	GVL_Modbus.modbusDamperInterface[2][1].enable     := TRUE;
	GVL_Modbus.modbusDamperInterface[2][2].enable     := TRUE;
	GVL_Modbus.modbusDamperInterface[2][3].enable     := TRUE;
	GVL_Modbus.modbusDamperInterface[2][4].enable     := TRUE;
	GVL_Modbus.modbusDamperInterface[2][5].enable     := TRUE;
	GVL_Modbus.modbusDamperInterface[2][6].enable     := TRUE;
	GVL_Modbus.modbusDamperInterface[2][7].enable     := TRUE;
	GVL_Modbus.modbusDamperInterface[2][8].enable     := TRUE;
	GVL_Modbus.modbusDamperInterface[2][9].enable     := TRUE;
	GVL_Modbus.modbusDamperInterface[2][10].enable     := TRUE;
	GVL_Modbus.modbusDamperInterface[2][11].enable     := TRUE;
	GVL_Modbus.modbusDamperInterface[2][12].enable     := TRUE;
	GVL_Modbus.modbusDamperInterface[2][13].enable     := TRUE;
	GVL_Modbus.modbusDamperInterface[2][14].enable     := TRUE;
	GVL_Modbus.modbusDamperInterface[2][15].enable     := TRUE;
	GVL_Modbus.modbusDamperInterface[2][16].enable     := TRUE;
	GVL_Modbus.modbusDamperInterface[2][17].enable     := TRUE;
	GVL_Modbus.modbusDamperInterface[2][18].enable     := TRUE;
	GVL_Modbus.modbusDamperInterface[2][19].enable     := TRUE;
	GVL_Modbus.modbusDamperInterface[2][20].enable     := TRUE;
	GVL_Modbus.modbusDamperInterface[2][21].enable     := TRUE;
	GVL_Modbus.modbusDamperInterface[2][22].enable     := TRUE;
	GVL_Modbus.modbusDamperInterface[2][23].enable     := TRUE;
	GVL_Modbus.modbusDamperInterface[2][24].enable     := TRUE;
	GVL_Modbus.modbusDamperInterface[2][25].enable     := TRUE;
	GVL_Modbus.modbusDamperInterface[2][26].enable     := TRUE;
	GVL_Modbus.modbusDamperInterface[2][1].systemNumber     := 01;
	GVL_Modbus.modbusDamperInterface[2][2].systemNumber     := 01;
	GVL_Modbus.modbusDamperInterface[2][3].systemNumber     := 01;
	GVL_Modbus.modbusDamperInterface[2][4].systemNumber     := 01;
	GVL_Modbus.modbusDamperInterface[2][5].systemNumber     := 01;
	GVL_Modbus.modbusDamperInterface[2][6].systemNumber     := 01;
	GVL_Modbus.modbusDamperInterface[2][7].systemNumber     := 01;
	GVL_Modbus.modbusDamperInterface[2][8].systemNumber     := 01;
	GVL_Modbus.modbusDamperInterface[2][9].systemNumber     := 01;
	GVL_Modbus.modbusDamperInterface[2][10].systemNumber     := 01;
	GVL_Modbus.modbusDamperInterface[2][11].systemNumber     := 01;
	GVL_Modbus.modbusDamperInterface[2][12].systemNumber     := 01;
	GVL_Modbus.modbusDamperInterface[2][13].systemNumber     := 01;
	GVL_Modbus.modbusDamperInterface[2][14].systemNumber     := 01;
	GVL_Modbus.modbusDamperInterface[2][15].systemNumber     := 01;
	GVL_Modbus.modbusDamperInterface[2][16].systemNumber     := 01;
	GVL_Modbus.modbusDamperInterface[2][17].systemNumber     := 01;
	GVL_Modbus.modbusDamperInterface[2][18].systemNumber     := 01;
	GVL_Modbus.modbusDamperInterface[2][19].systemNumber     := 01;
	GVL_Modbus.modbusDamperInterface[2][20].systemNumber     := 01;
	GVL_Modbus.modbusDamperInterface[2][21].systemNumber     := 01;
	GVL_Modbus.modbusDamperInterface[2][22].systemNumber     := 01;
	GVL_Modbus.modbusDamperInterface[2][23].systemNumber     := 01;
	GVL_Modbus.modbusDamperInterface[2][24].systemNumber     := 01;
	GVL_Modbus.modbusDamperInterface[2][25].systemNumber     := 01;
	GVL_Modbus.modbusDamperInterface[2][26].systemNumber     := 01;
	GVL_Modbus.modbusDamperInterface[2][1].systemPrefix     := 'A';
	GVL_Modbus.modbusDamperInterface[2][2].systemPrefix     := 'A';
	GVL_Modbus.modbusDamperInterface[2][3].systemPrefix     := 'A';
	GVL_Modbus.modbusDamperInterface[2][4].systemPrefix     := 'A';
	GVL_Modbus.modbusDamperInterface[2][5].systemPrefix     := 'A';
	GVL_Modbus.modbusDamperInterface[2][6].systemPrefix     := 'A';
	GVL_Modbus.modbusDamperInterface[2][7].systemPrefix     := 'A';
	GVL_Modbus.modbusDamperInterface[2][8].systemPrefix     := 'A';
	GVL_Modbus.modbusDamperInterface[2][9].systemPrefix     := 'A';
	GVL_Modbus.modbusDamperInterface[2][10].systemPrefix     := 'A';
	GVL_Modbus.modbusDamperInterface[2][11].systemPrefix     := 'A';
	GVL_Modbus.modbusDamperInterface[2][12].systemPrefix     := 'A';
	GVL_Modbus.modbusDamperInterface[2][13].systemPrefix     := 'A';
	GVL_Modbus.modbusDamperInterface[2][14].systemPrefix     := 'A';
	GVL_Modbus.modbusDamperInterface[2][15].systemPrefix     := 'A';
	GVL_Modbus.modbusDamperInterface[2][16].systemPrefix     := 'A';
	GVL_Modbus.modbusDamperInterface[2][17].systemPrefix     := 'A';
	GVL_Modbus.modbusDamperInterface[2][18].systemPrefix     := 'A';
	GVL_Modbus.modbusDamperInterface[2][19].systemPrefix     := 'A';
	GVL_Modbus.modbusDamperInterface[2][20].systemPrefix     := 'A';
	GVL_Modbus.modbusDamperInterface[2][21].systemPrefix     := 'A';
	GVL_Modbus.modbusDamperInterface[2][22].systemPrefix     := 'A';
	GVL_Modbus.modbusDamperInterface[2][23].systemPrefix     := 'A';
	GVL_Modbus.modbusDamperInterface[2][24].systemPrefix     := 'A';
	GVL_Modbus.modbusDamperInterface[2][25].systemPrefix     := 'A';
	GVL_Modbus.modbusDamperInterface[2][26].systemPrefix     := 'A';
	GVL_Modbus.modbusDamperInterface[2][1].airDirection     := 1;
	GVL_Modbus.modbusDamperInterface[2][2].airDirection     := 1;
	GVL_Modbus.modbusDamperInterface[2][3].airDirection     := 1;
	GVL_Modbus.modbusDamperInterface[2][4].airDirection     := 0;
	GVL_Modbus.modbusDamperInterface[2][5].airDirection     := 0;
	GVL_Modbus.modbusDamperInterface[2][6].airDirection     := 0;
	GVL_Modbus.modbusDamperInterface[2][7].airDirection     := 1;
	GVL_Modbus.modbusDamperInterface[2][8].airDirection     := 1;
	GVL_Modbus.modbusDamperInterface[2][9].airDirection     := 0;
	GVL_Modbus.modbusDamperInterface[2][10].airDirection     := 0;
	GVL_Modbus.modbusDamperInterface[2][11].airDirection     := 0;
	GVL_Modbus.modbusDamperInterface[2][12].airDirection     := 0;
	GVL_Modbus.modbusDamperInterface[2][13].airDirection     := 0;
	GVL_Modbus.modbusDamperInterface[2][14].airDirection     := 0;
	GVL_Modbus.modbusDamperInterface[2][15].airDirection     := 0;
	GVL_Modbus.modbusDamperInterface[2][16].airDirection     := 0;
	GVL_Modbus.modbusDamperInterface[2][17].airDirection     := 0;
	GVL_Modbus.modbusDamperInterface[2][18].airDirection     := 0;
	GVL_Modbus.modbusDamperInterface[2][19].airDirection     := 0;
	GVL_Modbus.modbusDamperInterface[2][20].airDirection     := 0;
	GVL_Modbus.modbusDamperInterface[2][21].airDirection     := 0;
	GVL_Modbus.modbusDamperInterface[2][22].airDirection     := 0;
	GVL_Modbus.modbusDamperInterface[2][23].airDirection     := 1;
	GVL_Modbus.modbusDamperInterface[2][24].airDirection     := 0;
	GVL_Modbus.modbusDamperInterface[2][25].airDirection     := 0;
	GVL_Modbus.modbusDamperInterface[2][26].airDirection     := 0;
	PersistentVars.ModbusDamperSetpoints[2][3].vMidM3h     := 100;
	PersistentVars.ModbusDamperSetpoints[2][9].vMidM3h     := 100;
	PersistentVars.ModbusDamperSetpoints[2][10].vMidM3h     := 100;
	PersistentVars.ModbusDamperSetpoints[2][11].vMidM3h     := 100;
	PersistentVars.ModbusDamperSetpoints[2][12].vMidM3h     := 100;
	PersistentVars.ModbusDamperSetpoints[2][13].vMidM3h     := 100;
	PersistentVars.ModbusDamperSetpoints[2][14].vMidM3h     := 100;
	PersistentVars.ModbusDamperSetpoints[2][15].vMidM3h     := 100;
	PersistentVars.ModbusDamperSetpoints[2][16].vMidM3h     := 100;
	PersistentVars.ModbusDamperSetpoints[2][17].vMidM3h     := 100;
	PersistentVars.ModbusDamperSetpoints[2][18].vMidM3h     := 160;
	PersistentVars.ModbusDamperSetpoints[2][19].vMidM3h     := 100;
	PersistentVars.ModbusDamperSetpoints[2][20].vMidM3h     := 100;
	PersistentVars.ModbusDamperSetpoints[2][21].vMidM3h     := 100;
	PersistentVars.ModbusDamperSetpoints[2][22].vMidM3h     := 100;
	PersistentVars.ModbusDamperSetpoints[2][24].vMidM3h     := 100;
	PersistentVars.ModbusDamperSetpoints[2][25].vMidM3h     := 100;
	PersistentVars.ModbusDamperSetpoints[2][26].vMidM3h     := 100;
                            
                        
END_ACTION
END_PROGRAM

PROGRAM PRG_DamperLine_3

                
    
	if (firstScan) then
	    initialSettings();
	end_if
	
	GVL_Modbus.modbusDamperInterface[3][1].tag     := 'B=360.02-SQ5UBH1';
	GVL_Modbus.modbusDamperInterface[3][2].tag     := 'B=360.02-SQ5UBH2';
	GVL_Modbus.modbusDamperInterface[3][3].tag     := 'B=360.02-SQ4UBH1';
	GVL_Modbus.modbusDamperInterface[3][4].tag     := 'B=360.02-SQ4UBH2';
	GVL_Modbus.modbusDamperInterface[3][1].damperClimateInterface     := GVL_ClimateControl.typClimateControllerInterfaceRoomSONE.actuators.damper;
	GVL_Modbus.modbusDamperInterface[3][2].damperClimateInterface     := GVL_ClimateControl.typClimateControllerInterfaceRoomSONE.actuators.damper;
	GVL_Modbus.modbusDamperInterface[3][3].damperClimateInterface     := GVL_ClimateControl.typClimateControllerInterfaceRoomSONE.actuators.damper;
	GVL_Modbus.modbusDamperInterface[3][4].damperClimateInterface     := GVL_ClimateControl.typClimateControllerInterfaceRoomSONE.actuators.damper;
                
              

ACTION initialSettings:
                            
                                
	GVL_Modbus.modbusDamperInterface[3][1].enable     := TRUE;
	GVL_Modbus.modbusDamperInterface[3][2].enable     := TRUE;
	GVL_Modbus.modbusDamperInterface[3][3].enable     := TRUE;
	GVL_Modbus.modbusDamperInterface[3][4].enable     := TRUE;
	GVL_Modbus.modbusDamperInterface[3][1].systemNumber     := 02;
	GVL_Modbus.modbusDamperInterface[3][2].systemNumber     := 02;
	GVL_Modbus.modbusDamperInterface[3][3].systemNumber     := 02;
	GVL_Modbus.modbusDamperInterface[3][4].systemNumber     := 02;
	GVL_Modbus.modbusDamperInterface[3][1].systemPrefix     := 'B';
	GVL_Modbus.modbusDamperInterface[3][2].systemPrefix     := 'B';
	GVL_Modbus.modbusDamperInterface[3][3].systemPrefix     := 'B';
	GVL_Modbus.modbusDamperInterface[3][4].systemPrefix     := 'B';
	GVL_Modbus.modbusDamperInterface[3][1].airDirection     := 1;
	GVL_Modbus.modbusDamperInterface[3][2].airDirection     := 1;
	GVL_Modbus.modbusDamperInterface[3][3].airDirection     := 0;
	GVL_Modbus.modbusDamperInterface[3][4].airDirection     := 0;
                            
                        
END_ACTION
END_PROGRAM

PROGRAM PRG_StateTexts

                
    
	IF (firstScan) THEN
C_5640_501_06_RTC01_MOD_FB_R0401.setStateText(1, 'Frostbeskyttelse');
C_5640_501_06_RTC01_MOD_FB_R0401.setStateText(2, 'Økonomi');
C_5640_501_06_RTC01_MOD_FB_R0401.setStateText(3, 'Standby');
C_5640_501_06_RTC01_MOD_FB_R0401.setStateText(4, 'Komfort');
C_5640_501_06_RTC01_MOD_FB_R0401.setStateText(5, 'Nattkjøling');
C_5640_501_06_RTC01_KMD_MSV_R0401.setStateText(1, 'Kalender 1');
C_5640_501_06_RTC01_KMD_MSV_R0401.setStateText(2, 'Kalender 2');
C_5640_501_06_RTC01_KMD_MSV_R0401.setStateText(3, 'Kalender 3');
C_5640_501_06_RTC01_KMD_MSV_R0401.setStateText(4, 'Kalender 4');
C_5640_501_06_RTC01_KMD_MSV_R0401.setStateText(5, 'Kalender 5');
C_5640_501_06_RTC01_KMD_MSV_R0401.setStateText(6, 'Kalender 6');
C_5640_501_06_RTC01_KMD_MSV_R0401.setStateText(7, 'Kalender 7');
C_5640_501_06_RTC01_KMD_MSV_R0401.setStateText(8, 'Kalender 8');
C_5640_501_06_RTC01_KMD_MSV_R0401.setStateText(9, 'Kalender 9');
C_5640_501_06_RTC01_KMD_MSV_R0401.setStateText(10, 'Kalender 10');
C_5640_501_06_RTC01_MOD_FB_R0406.setStateText(1, 'Frostbeskyttelse');
C_5640_501_06_RTC01_MOD_FB_R0406.setStateText(2, 'Økonomi');
C_5640_501_06_RTC01_MOD_FB_R0406.setStateText(3, 'Standby');
C_5640_501_06_RTC01_MOD_FB_R0406.setStateText(4, 'Komfort');
C_5640_501_06_RTC01_MOD_FB_R0406.setStateText(5, 'Nattkjøling');
C_5640_501_06_RTC01_KMD_MSV_R0406.setStateText(1, 'Kalender 1');
C_5640_501_06_RTC01_KMD_MSV_R0406.setStateText(2, 'Kalender 2');
C_5640_501_06_RTC01_KMD_MSV_R0406.setStateText(3, 'Kalender 3');
C_5640_501_06_RTC01_KMD_MSV_R0406.setStateText(4, 'Kalender 4');
C_5640_501_06_RTC01_KMD_MSV_R0406.setStateText(5, 'Kalender 5');
C_5640_501_06_RTC01_KMD_MSV_R0406.setStateText(6, 'Kalender 6');
C_5640_501_06_RTC01_KMD_MSV_R0406.setStateText(7, 'Kalender 7');
C_5640_501_06_RTC01_KMD_MSV_R0406.setStateText(8, 'Kalender 8');
C_5640_501_06_RTC01_KMD_MSV_R0406.setStateText(9, 'Kalender 9');
C_5640_501_06_RTC01_KMD_MSV_R0406.setStateText(10, 'Kalender 10');
C_5640_501_06_RTC01_MOD_FB_R0407.setStateText(1, 'Frostbeskyttelse');
C_5640_501_06_RTC01_MOD_FB_R0407.setStateText(2, 'Økonomi');
C_5640_501_06_RTC01_MOD_FB_R0407.setStateText(3, 'Standby');
C_5640_501_06_RTC01_MOD_FB_R0407.setStateText(4, 'Komfort');
C_5640_501_06_RTC01_MOD_FB_R0407.setStateText(5, 'Nattkjøling');
C_5640_501_06_RTC01_KMD_MSV_R0407.setStateText(1, 'Kalender 1');
C_5640_501_06_RTC01_KMD_MSV_R0407.setStateText(2, 'Kalender 2');
C_5640_501_06_RTC01_KMD_MSV_R0407.setStateText(3, 'Kalender 3');
C_5640_501_06_RTC01_KMD_MSV_R0407.setStateText(4, 'Kalender 4');
C_5640_501_06_RTC01_KMD_MSV_R0407.setStateText(5, 'Kalender 5');
C_5640_501_06_RTC01_KMD_MSV_R0407.setStateText(6, 'Kalender 6');
C_5640_501_06_RTC01_KMD_MSV_R0407.setStateText(7, 'Kalender 7');
C_5640_501_06_RTC01_KMD_MSV_R0407.setStateText(8, 'Kalender 8');
C_5640_501_06_RTC01_KMD_MSV_R0407.setStateText(9, 'Kalender 9');
C_5640_501_06_RTC01_KMD_MSV_R0407.setStateText(10, 'Kalender 10');
C_5640_501_06_RTC01_MOD_FB_R0408.setStateText(1, 'Frostbeskyttelse');
C_5640_501_06_RTC01_MOD_FB_R0408.setStateText(2, 'Økonomi');
C_5640_501_06_RTC01_MOD_FB_R0408.setStateText(3, 'Standby');
C_5640_501_06_RTC01_MOD_FB_R0408.setStateText(4, 'Komfort');
C_5640_501_06_RTC01_MOD_FB_R0408.setStateText(5, 'Nattkjøling');
C_5640_501_06_RTC01_KMD_MSV_R0408.setStateText(1, 'Kalender 1');
C_5640_501_06_RTC01_KMD_MSV_R0408.setStateText(2, 'Kalender 2');
C_5640_501_06_RTC01_KMD_MSV_R0408.setStateText(3, 'Kalender 3');
C_5640_501_06_RTC01_KMD_MSV_R0408.setStateText(4, 'Kalender 4');
C_5640_501_06_RTC01_KMD_MSV_R0408.setStateText(5, 'Kalender 5');
C_5640_501_06_RTC01_KMD_MSV_R0408.setStateText(6, 'Kalender 6');
C_5640_501_06_RTC01_KMD_MSV_R0408.setStateText(7, 'Kalender 7');
C_5640_501_06_RTC01_KMD_MSV_R0408.setStateText(8, 'Kalender 8');
C_5640_501_06_RTC01_KMD_MSV_R0408.setStateText(9, 'Kalender 9');
C_5640_501_06_RTC01_KMD_MSV_R0408.setStateText(10, 'Kalender 10');
C_5640_501_06_RTC01_MOD_FB_R0409.setStateText(1, 'Frostbeskyttelse');
C_5640_501_06_RTC01_MOD_FB_R0409.setStateText(2, 'Økonomi');
C_5640_501_06_RTC01_MOD_FB_R0409.setStateText(3, 'Standby');
C_5640_501_06_RTC01_MOD_FB_R0409.setStateText(4, 'Komfort');
C_5640_501_06_RTC01_MOD_FB_R0409.setStateText(5, 'Nattkjøling');
C_5640_501_06_RTC01_KMD_MSV_R0409.setStateText(1, 'Kalender 1');
C_5640_501_06_RTC01_KMD_MSV_R0409.setStateText(2, 'Kalender 2');
C_5640_501_06_RTC01_KMD_MSV_R0409.setStateText(3, 'Kalender 3');
C_5640_501_06_RTC01_KMD_MSV_R0409.setStateText(4, 'Kalender 4');
C_5640_501_06_RTC01_KMD_MSV_R0409.setStateText(5, 'Kalender 5');
C_5640_501_06_RTC01_KMD_MSV_R0409.setStateText(6, 'Kalender 6');
C_5640_501_06_RTC01_KMD_MSV_R0409.setStateText(7, 'Kalender 7');
C_5640_501_06_RTC01_KMD_MSV_R0409.setStateText(8, 'Kalender 8');
C_5640_501_06_RTC01_KMD_MSV_R0409.setStateText(9, 'Kalender 9');
C_5640_501_06_RTC01_KMD_MSV_R0409.setStateText(10, 'Kalender 10');
C_5640_501_06_RTC01_MOD_FB_R0464.setStateText(1, 'Frostbeskyttelse');
C_5640_501_06_RTC01_MOD_FB_R0464.setStateText(2, 'Økonomi');
C_5640_501_06_RTC01_MOD_FB_R0464.setStateText(3, 'Standby');
C_5640_501_06_RTC01_MOD_FB_R0464.setStateText(4, 'Komfort');
C_5640_501_06_RTC01_MOD_FB_R0464.setStateText(5, 'Nattkjøling');
C_5640_501_06_RTC01_KMD_MSV_R0464.setStateText(1, 'Kalender 1');
C_5640_501_06_RTC01_KMD_MSV_R0464.setStateText(2, 'Kalender 2');
C_5640_501_06_RTC01_KMD_MSV_R0464.setStateText(3, 'Kalender 3');
C_5640_501_06_RTC01_KMD_MSV_R0464.setStateText(4, 'Kalender 4');
C_5640_501_06_RTC01_KMD_MSV_R0464.setStateText(5, 'Kalender 5');
C_5640_501_06_RTC01_KMD_MSV_R0464.setStateText(6, 'Kalender 6');
C_5640_501_06_RTC01_KMD_MSV_R0464.setStateText(7, 'Kalender 7');
C_5640_501_06_RTC01_KMD_MSV_R0464.setStateText(8, 'Kalender 8');
C_5640_501_06_RTC01_KMD_MSV_R0464.setStateText(9, 'Kalender 9');
C_5640_501_06_RTC01_KMD_MSV_R0464.setStateText(10, 'Kalender 10');
C_5640_501_06_RTC01_MOD_FB_R0415.setStateText(1, 'Frostbeskyttelse');
C_5640_501_06_RTC01_MOD_FB_R0415.setStateText(2, 'Økonomi');
C_5640_501_06_RTC01_MOD_FB_R0415.setStateText(3, 'Standby');
C_5640_501_06_RTC01_MOD_FB_R0415.setStateText(4, 'Komfort');
C_5640_501_06_RTC01_MOD_FB_R0415.setStateText(5, 'Nattkjøling');
C_5640_501_06_RTC01_KMD_MSV_R0415.setStateText(1, 'Kalender 1');
C_5640_501_06_RTC01_KMD_MSV_R0415.setStateText(2, 'Kalender 2');
C_5640_501_06_RTC01_KMD_MSV_R0415.setStateText(3, 'Kalender 3');
C_5640_501_06_RTC01_KMD_MSV_R0415.setStateText(4, 'Kalender 4');
C_5640_501_06_RTC01_KMD_MSV_R0415.setStateText(5, 'Kalender 5');
C_5640_501_06_RTC01_KMD_MSV_R0415.setStateText(6, 'Kalender 6');
C_5640_501_06_RTC01_KMD_MSV_R0415.setStateText(7, 'Kalender 7');
C_5640_501_06_RTC01_KMD_MSV_R0415.setStateText(8, 'Kalender 8');
C_5640_501_06_RTC01_KMD_MSV_R0415.setStateText(9, 'Kalender 9');
C_5640_501_06_RTC01_KMD_MSV_R0415.setStateText(10, 'Kalender 10');
C_5640_501_06_RTC01_MOD_FB_R0422.setStateText(1, 'Frostbeskyttelse');
C_5640_501_06_RTC01_MOD_FB_R0422.setStateText(2, 'Økonomi');
C_5640_501_06_RTC01_MOD_FB_R0422.setStateText(3, 'Standby');
C_5640_501_06_RTC01_MOD_FB_R0422.setStateText(4, 'Komfort');
C_5640_501_06_RTC01_MOD_FB_R0422.setStateText(5, 'Nattkjøling');
C_5640_501_06_RTC01_KMD_MSV_R0422.setStateText(1, 'Kalender 1');
C_5640_501_06_RTC01_KMD_MSV_R0422.setStateText(2, 'Kalender 2');
C_5640_501_06_RTC01_KMD_MSV_R0422.setStateText(3, 'Kalender 3');
C_5640_501_06_RTC01_KMD_MSV_R0422.setStateText(4, 'Kalender 4');
C_5640_501_06_RTC01_KMD_MSV_R0422.setStateText(5, 'Kalender 5');
C_5640_501_06_RTC01_KMD_MSV_R0422.setStateText(6, 'Kalender 6');
C_5640_501_06_RTC01_KMD_MSV_R0422.setStateText(7, 'Kalender 7');
C_5640_501_06_RTC01_KMD_MSV_R0422.setStateText(8, 'Kalender 8');
C_5640_501_06_RTC01_KMD_MSV_R0422.setStateText(9, 'Kalender 9');
C_5640_501_06_RTC01_KMD_MSV_R0422.setStateText(10, 'Kalender 10');
C_5640_501_06_RTC01_MOD_FB_R0426_1.setStateText(1, 'Frostbeskyttelse');
C_5640_501_06_RTC01_MOD_FB_R0426_1.setStateText(2, 'Økonomi');
C_5640_501_06_RTC01_MOD_FB_R0426_1.setStateText(3, 'Standby');
C_5640_501_06_RTC01_MOD_FB_R0426_1.setStateText(4, 'Komfort');
C_5640_501_06_RTC01_MOD_FB_R0426_1.setStateText(5, 'Nattkjøling');
C_5640_501_06_RTC01_KMD_MSV_R0426_1.setStateText(1, 'Kalender 1');
C_5640_501_06_RTC01_KMD_MSV_R0426_1.setStateText(2, 'Kalender 2');
C_5640_501_06_RTC01_KMD_MSV_R0426_1.setStateText(3, 'Kalender 3');
C_5640_501_06_RTC01_KMD_MSV_R0426_1.setStateText(4, 'Kalender 4');
C_5640_501_06_RTC01_KMD_MSV_R0426_1.setStateText(5, 'Kalender 5');
C_5640_501_06_RTC01_KMD_MSV_R0426_1.setStateText(6, 'Kalender 6');
C_5640_501_06_RTC01_KMD_MSV_R0426_1.setStateText(7, 'Kalender 7');
C_5640_501_06_RTC01_KMD_MSV_R0426_1.setStateText(8, 'Kalender 8');
C_5640_501_06_RTC01_KMD_MSV_R0426_1.setStateText(9, 'Kalender 9');
C_5640_501_06_RTC01_KMD_MSV_R0426_1.setStateText(10, 'Kalender 10');
C_5640_501_06_RTC01_MOD_FB_R0426_2.setStateText(1, 'Frostbeskyttelse');
C_5640_501_06_RTC01_MOD_FB_R0426_2.setStateText(2, 'Økonomi');
C_5640_501_06_RTC01_MOD_FB_R0426_2.setStateText(3, 'Standby');
C_5640_501_06_RTC01_MOD_FB_R0426_2.setStateText(4, 'Komfort');
C_5640_501_06_RTC01_MOD_FB_R0426_2.setStateText(5, 'Nattkjøling');
C_5640_501_06_RTC01_KMD_MSV_R0426_2.setStateText(1, 'Kalender 1');
C_5640_501_06_RTC01_KMD_MSV_R0426_2.setStateText(2, 'Kalender 2');
C_5640_501_06_RTC01_KMD_MSV_R0426_2.setStateText(3, 'Kalender 3');
C_5640_501_06_RTC01_KMD_MSV_R0426_2.setStateText(4, 'Kalender 4');
C_5640_501_06_RTC01_KMD_MSV_R0426_2.setStateText(5, 'Kalender 5');
C_5640_501_06_RTC01_KMD_MSV_R0426_2.setStateText(6, 'Kalender 6');
C_5640_501_06_RTC01_KMD_MSV_R0426_2.setStateText(7, 'Kalender 7');
C_5640_501_06_RTC01_KMD_MSV_R0426_2.setStateText(8, 'Kalender 8');
C_5640_501_06_RTC01_KMD_MSV_R0426_2.setStateText(9, 'Kalender 9');
C_5640_501_06_RTC01_KMD_MSV_R0426_2.setStateText(10, 'Kalender 10');
C_5640_501_06_RTC01_MOD_FB_R0426_3.setStateText(1, 'Frostbeskyttelse');
C_5640_501_06_RTC01_MOD_FB_R0426_3.setStateText(2, 'Økonomi');
C_5640_501_06_RTC01_MOD_FB_R0426_3.setStateText(3, 'Standby');
C_5640_501_06_RTC01_MOD_FB_R0426_3.setStateText(4, 'Komfort');
C_5640_501_06_RTC01_MOD_FB_R0426_3.setStateText(5, 'Nattkjøling');
C_5640_501_06_RTC01_KMD_MSV_R0426_3.setStateText(1, 'Kalender 1');
C_5640_501_06_RTC01_KMD_MSV_R0426_3.setStateText(2, 'Kalender 2');
C_5640_501_06_RTC01_KMD_MSV_R0426_3.setStateText(3, 'Kalender 3');
C_5640_501_06_RTC01_KMD_MSV_R0426_3.setStateText(4, 'Kalender 4');
C_5640_501_06_RTC01_KMD_MSV_R0426_3.setStateText(5, 'Kalender 5');
C_5640_501_06_RTC01_KMD_MSV_R0426_3.setStateText(6, 'Kalender 6');
C_5640_501_06_RTC01_KMD_MSV_R0426_3.setStateText(7, 'Kalender 7');
C_5640_501_06_RTC01_KMD_MSV_R0426_3.setStateText(8, 'Kalender 8');
C_5640_501_06_RTC01_KMD_MSV_R0426_3.setStateText(9, 'Kalender 9');
C_5640_501_06_RTC01_KMD_MSV_R0426_3.setStateText(10, 'Kalender 10');
C_5640_501_06_RTC01_MOD_FB_R0528.setStateText(1, 'Frostbeskyttelse');
C_5640_501_06_RTC01_MOD_FB_R0528.setStateText(2, 'Økonomi');
C_5640_501_06_RTC01_MOD_FB_R0528.setStateText(3, 'Standby');
C_5640_501_06_RTC01_MOD_FB_R0528.setStateText(4, 'Komfort');
C_5640_501_06_RTC01_MOD_FB_R0528.setStateText(5, 'Nattkjøling');
C_5640_501_06_RTC01_KMD_MSV_R0528.setStateText(1, 'Kalender 1');
C_5640_501_06_RTC01_KMD_MSV_R0528.setStateText(2, 'Kalender 2');
C_5640_501_06_RTC01_KMD_MSV_R0528.setStateText(3, 'Kalender 3');
C_5640_501_06_RTC01_KMD_MSV_R0528.setStateText(4, 'Kalender 4');
C_5640_501_06_RTC01_KMD_MSV_R0528.setStateText(5, 'Kalender 5');
C_5640_501_06_RTC01_KMD_MSV_R0528.setStateText(6, 'Kalender 6');
C_5640_501_06_RTC01_KMD_MSV_R0528.setStateText(7, 'Kalender 7');
C_5640_501_06_RTC01_KMD_MSV_R0528.setStateText(8, 'Kalender 8');
C_5640_501_06_RTC01_KMD_MSV_R0528.setStateText(9, 'Kalender 9');
C_5640_501_06_RTC01_KMD_MSV_R0528.setStateText(10, 'Kalender 10');
C_5640_501_06_RTC01_MOD_FB_R0523.setStateText(1, 'Frostbeskyttelse');
C_5640_501_06_RTC01_MOD_FB_R0523.setStateText(2, 'Økonomi');
C_5640_501_06_RTC01_MOD_FB_R0523.setStateText(3, 'Standby');
C_5640_501_06_RTC01_MOD_FB_R0523.setStateText(4, 'Komfort');
C_5640_501_06_RTC01_MOD_FB_R0523.setStateText(5, 'Nattkjøling');
C_5640_501_06_RTC01_KMD_MSV_R0523.setStateText(1, 'Kalender 1');
C_5640_501_06_RTC01_KMD_MSV_R0523.setStateText(2, 'Kalender 2');
C_5640_501_06_RTC01_KMD_MSV_R0523.setStateText(3, 'Kalender 3');
C_5640_501_06_RTC01_KMD_MSV_R0523.setStateText(4, 'Kalender 4');
C_5640_501_06_RTC01_KMD_MSV_R0523.setStateText(5, 'Kalender 5');
C_5640_501_06_RTC01_KMD_MSV_R0523.setStateText(6, 'Kalender 6');
C_5640_501_06_RTC01_KMD_MSV_R0523.setStateText(7, 'Kalender 7');
C_5640_501_06_RTC01_KMD_MSV_R0523.setStateText(8, 'Kalender 8');
C_5640_501_06_RTC01_KMD_MSV_R0523.setStateText(9, 'Kalender 9');
C_5640_501_06_RTC01_KMD_MSV_R0523.setStateText(10, 'Kalender 10');
C_5640_501_06_RTC01_MOD_FB_R0531.setStateText(1, 'Frostbeskyttelse');
C_5640_501_06_RTC01_MOD_FB_R0531.setStateText(2, 'Økonomi');
C_5640_501_06_RTC01_MOD_FB_R0531.setStateText(3, 'Standby');
C_5640_501_06_RTC01_MOD_FB_R0531.setStateText(4, 'Komfort');
C_5640_501_06_RTC01_MOD_FB_R0531.setStateText(5, 'Nattkjøling');
C_5640_501_06_RTC01_KMD_MSV_R0531.setStateText(1, 'Kalender 1');
C_5640_501_06_RTC01_KMD_MSV_R0531.setStateText(2, 'Kalender 2');
C_5640_501_06_RTC01_KMD_MSV_R0531.setStateText(3, 'Kalender 3');
C_5640_501_06_RTC01_KMD_MSV_R0531.setStateText(4, 'Kalender 4');
C_5640_501_06_RTC01_KMD_MSV_R0531.setStateText(5, 'Kalender 5');
C_5640_501_06_RTC01_KMD_MSV_R0531.setStateText(6, 'Kalender 6');
C_5640_501_06_RTC01_KMD_MSV_R0531.setStateText(7, 'Kalender 7');
C_5640_501_06_RTC01_KMD_MSV_R0531.setStateText(8, 'Kalender 8');
C_5640_501_06_RTC01_KMD_MSV_R0531.setStateText(9, 'Kalender 9');
C_5640_501_06_RTC01_KMD_MSV_R0531.setStateText(10, 'Kalender 10');
C_5640_501_06_RTC01_MOD_FB_R0535_1.setStateText(1, 'Frostbeskyttelse');
C_5640_501_06_RTC01_MOD_FB_R0535_1.setStateText(2, 'Økonomi');
C_5640_501_06_RTC01_MOD_FB_R0535_1.setStateText(3, 'Standby');
C_5640_501_06_RTC01_MOD_FB_R0535_1.setStateText(4, 'Komfort');
C_5640_501_06_RTC01_MOD_FB_R0535_1.setStateText(5, 'Nattkjøling');
C_5640_501_06_RTC01_KMD_MSV_R0535_1.setStateText(1, 'Kalender 1');
C_5640_501_06_RTC01_KMD_MSV_R0535_1.setStateText(2, 'Kalender 2');
C_5640_501_06_RTC01_KMD_MSV_R0535_1.setStateText(3, 'Kalender 3');
C_5640_501_06_RTC01_KMD_MSV_R0535_1.setStateText(4, 'Kalender 4');
C_5640_501_06_RTC01_KMD_MSV_R0535_1.setStateText(5, 'Kalender 5');
C_5640_501_06_RTC01_KMD_MSV_R0535_1.setStateText(6, 'Kalender 6');
C_5640_501_06_RTC01_KMD_MSV_R0535_1.setStateText(7, 'Kalender 7');
C_5640_501_06_RTC01_KMD_MSV_R0535_1.setStateText(8, 'Kalender 8');
C_5640_501_06_RTC01_KMD_MSV_R0535_1.setStateText(9, 'Kalender 9');
C_5640_501_06_RTC01_KMD_MSV_R0535_1.setStateText(10, 'Kalender 10');
C_5640_501_06_RTC01_MOD_FB_R0535_2.setStateText(1, 'Frostbeskyttelse');
C_5640_501_06_RTC01_MOD_FB_R0535_2.setStateText(2, 'Økonomi');
C_5640_501_06_RTC01_MOD_FB_R0535_2.setStateText(3, 'Standby');
C_5640_501_06_RTC01_MOD_FB_R0535_2.setStateText(4, 'Komfort');
C_5640_501_06_RTC01_MOD_FB_R0535_2.setStateText(5, 'Nattkjøling');
C_5640_501_06_RTC01_KMD_MSV_R0535_2.setStateText(1, 'Kalender 1');
C_5640_501_06_RTC01_KMD_MSV_R0535_2.setStateText(2, 'Kalender 2');
C_5640_501_06_RTC01_KMD_MSV_R0535_2.setStateText(3, 'Kalender 3');
C_5640_501_06_RTC01_KMD_MSV_R0535_2.setStateText(4, 'Kalender 4');
C_5640_501_06_RTC01_KMD_MSV_R0535_2.setStateText(5, 'Kalender 5');
C_5640_501_06_RTC01_KMD_MSV_R0535_2.setStateText(6, 'Kalender 6');
C_5640_501_06_RTC01_KMD_MSV_R0535_2.setStateText(7, 'Kalender 7');
C_5640_501_06_RTC01_KMD_MSV_R0535_2.setStateText(8, 'Kalender 8');
C_5640_501_06_RTC01_KMD_MSV_R0535_2.setStateText(9, 'Kalender 9');
C_5640_501_06_RTC01_KMD_MSV_R0535_2.setStateText(10, 'Kalender 10');
C_5640_501_06_RTC01_MOD_FB_R0535_3.setStateText(1, 'Frostbeskyttelse');
C_5640_501_06_RTC01_MOD_FB_R0535_3.setStateText(2, 'Økonomi');
C_5640_501_06_RTC01_MOD_FB_R0535_3.setStateText(3, 'Standby');
C_5640_501_06_RTC01_MOD_FB_R0535_3.setStateText(4, 'Komfort');
C_5640_501_06_RTC01_MOD_FB_R0535_3.setStateText(5, 'Nattkjøling');
C_5640_501_06_RTC01_KMD_MSV_R0535_3.setStateText(1, 'Kalender 1');
C_5640_501_06_RTC01_KMD_MSV_R0535_3.setStateText(2, 'Kalender 2');
C_5640_501_06_RTC01_KMD_MSV_R0535_3.setStateText(3, 'Kalender 3');
C_5640_501_06_RTC01_KMD_MSV_R0535_3.setStateText(4, 'Kalender 4');
C_5640_501_06_RTC01_KMD_MSV_R0535_3.setStateText(5, 'Kalender 5');
C_5640_501_06_RTC01_KMD_MSV_R0535_3.setStateText(6, 'Kalender 6');
C_5640_501_06_RTC01_KMD_MSV_R0535_3.setStateText(7, 'Kalender 7');
C_5640_501_06_RTC01_KMD_MSV_R0535_3.setStateText(8, 'Kalender 8');
C_5640_501_06_RTC01_KMD_MSV_R0535_3.setStateText(9, 'Kalender 9');
C_5640_501_06_RTC01_KMD_MSV_R0535_3.setStateText(10, 'Kalender 10');
C_5640_501_06_RTC01_MOD_FB_R0536.setStateText(1, 'Frostbeskyttelse');
C_5640_501_06_RTC01_MOD_FB_R0536.setStateText(2, 'Økonomi');
C_5640_501_06_RTC01_MOD_FB_R0536.setStateText(3, 'Standby');
C_5640_501_06_RTC01_MOD_FB_R0536.setStateText(4, 'Komfort');
C_5640_501_06_RTC01_MOD_FB_R0536.setStateText(5, 'Nattkjøling');
C_5640_501_06_RTC01_KMD_MSV_R0536.setStateText(1, 'Kalender 1');
C_5640_501_06_RTC01_KMD_MSV_R0536.setStateText(2, 'Kalender 2');
C_5640_501_06_RTC01_KMD_MSV_R0536.setStateText(3, 'Kalender 3');
C_5640_501_06_RTC01_KMD_MSV_R0536.setStateText(4, 'Kalender 4');
C_5640_501_06_RTC01_KMD_MSV_R0536.setStateText(5, 'Kalender 5');
C_5640_501_06_RTC01_KMD_MSV_R0536.setStateText(6, 'Kalender 6');
C_5640_501_06_RTC01_KMD_MSV_R0536.setStateText(7, 'Kalender 7');
C_5640_501_06_RTC01_KMD_MSV_R0536.setStateText(8, 'Kalender 8');
C_5640_501_06_RTC01_KMD_MSV_R0536.setStateText(9, 'Kalender 9');
C_5640_501_06_RTC01_KMD_MSV_R0536.setStateText(10, 'Kalender 10');
C_5640_501_06_RTC01_MOD_FB_R0543.setStateText(1, 'Frostbeskyttelse');
C_5640_501_06_RTC01_MOD_FB_R0543.setStateText(2, 'Økonomi');
C_5640_501_06_RTC01_MOD_FB_R0543.setStateText(3, 'Standby');
C_5640_501_06_RTC01_MOD_FB_R0543.setStateText(4, 'Komfort');
C_5640_501_06_RTC01_MOD_FB_R0543.setStateText(5, 'Nattkjøling');
C_5640_501_06_RTC01_KMD_MSV_R0543.setStateText(1, 'Kalender 1');
C_5640_501_06_RTC01_KMD_MSV_R0543.setStateText(2, 'Kalender 2');
C_5640_501_06_RTC01_KMD_MSV_R0543.setStateText(3, 'Kalender 3');
C_5640_501_06_RTC01_KMD_MSV_R0543.setStateText(4, 'Kalender 4');
C_5640_501_06_RTC01_KMD_MSV_R0543.setStateText(5, 'Kalender 5');
C_5640_501_06_RTC01_KMD_MSV_R0543.setStateText(6, 'Kalender 6');
C_5640_501_06_RTC01_KMD_MSV_R0543.setStateText(7, 'Kalender 7');
C_5640_501_06_RTC01_KMD_MSV_R0543.setStateText(8, 'Kalender 8');
C_5640_501_06_RTC01_KMD_MSV_R0543.setStateText(9, 'Kalender 9');
C_5640_501_06_RTC01_KMD_MSV_R0543.setStateText(10, 'Kalender 10');
C_5640_501_06_RTC01_MOD_FB_R0547_1.setStateText(1, 'Frostbeskyttelse');
C_5640_501_06_RTC01_MOD_FB_R0547_1.setStateText(2, 'Økonomi');
C_5640_501_06_RTC01_MOD_FB_R0547_1.setStateText(3, 'Standby');
C_5640_501_06_RTC01_MOD_FB_R0547_1.setStateText(4, 'Komfort');
C_5640_501_06_RTC01_MOD_FB_R0547_1.setStateText(5, 'Nattkjøling');
C_5640_501_06_RTC01_KMD_MSV_R0547_1.setStateText(1, 'Kalender 1');
C_5640_501_06_RTC01_KMD_MSV_R0547_1.setStateText(2, 'Kalender 2');
C_5640_501_06_RTC01_KMD_MSV_R0547_1.setStateText(3, 'Kalender 3');
C_5640_501_06_RTC01_KMD_MSV_R0547_1.setStateText(4, 'Kalender 4');
C_5640_501_06_RTC01_KMD_MSV_R0547_1.setStateText(5, 'Kalender 5');
C_5640_501_06_RTC01_KMD_MSV_R0547_1.setStateText(6, 'Kalender 6');
C_5640_501_06_RTC01_KMD_MSV_R0547_1.setStateText(7, 'Kalender 7');
C_5640_501_06_RTC01_KMD_MSV_R0547_1.setStateText(8, 'Kalender 8');
C_5640_501_06_RTC01_KMD_MSV_R0547_1.setStateText(9, 'Kalender 9');
C_5640_501_06_RTC01_KMD_MSV_R0547_1.setStateText(10, 'Kalender 10');
C_5640_501_06_RTC01_MOD_FB_R0547_2.setStateText(1, 'Frostbeskyttelse');
C_5640_501_06_RTC01_MOD_FB_R0547_2.setStateText(2, 'Økonomi');
C_5640_501_06_RTC01_MOD_FB_R0547_2.setStateText(3, 'Standby');
C_5640_501_06_RTC01_MOD_FB_R0547_2.setStateText(4, 'Komfort');
C_5640_501_06_RTC01_MOD_FB_R0547_2.setStateText(5, 'Nattkjøling');
C_5640_501_06_RTC01_KMD_MSV_R0547_2.setStateText(1, 'Kalender 1');
C_5640_501_06_RTC01_KMD_MSV_R0547_2.setStateText(2, 'Kalender 2');
C_5640_501_06_RTC01_KMD_MSV_R0547_2.setStateText(3, 'Kalender 3');
C_5640_501_06_RTC01_KMD_MSV_R0547_2.setStateText(4, 'Kalender 4');
C_5640_501_06_RTC01_KMD_MSV_R0547_2.setStateText(5, 'Kalender 5');
C_5640_501_06_RTC01_KMD_MSV_R0547_2.setStateText(6, 'Kalender 6');
C_5640_501_06_RTC01_KMD_MSV_R0547_2.setStateText(7, 'Kalender 7');
C_5640_501_06_RTC01_KMD_MSV_R0547_2.setStateText(8, 'Kalender 8');
C_5640_501_06_RTC01_KMD_MSV_R0547_2.setStateText(9, 'Kalender 9');
C_5640_501_06_RTC01_KMD_MSV_R0547_2.setStateText(10, 'Kalender 10');
C_5640_501_06_RTC01_MOD_FB_R0544.setStateText(1, 'Frostbeskyttelse');
C_5640_501_06_RTC01_MOD_FB_R0544.setStateText(2, 'Økonomi');
C_5640_501_06_RTC01_MOD_FB_R0544.setStateText(3, 'Standby');
C_5640_501_06_RTC01_MOD_FB_R0544.setStateText(4, 'Komfort');
C_5640_501_06_RTC01_MOD_FB_R0544.setStateText(5, 'Nattkjøling');
C_5640_501_06_RTC01_KMD_MSV_R0544.setStateText(1, 'Kalender 1');
C_5640_501_06_RTC01_KMD_MSV_R0544.setStateText(2, 'Kalender 2');
C_5640_501_06_RTC01_KMD_MSV_R0544.setStateText(3, 'Kalender 3');
C_5640_501_06_RTC01_KMD_MSV_R0544.setStateText(4, 'Kalender 4');
C_5640_501_06_RTC01_KMD_MSV_R0544.setStateText(5, 'Kalender 5');
C_5640_501_06_RTC01_KMD_MSV_R0544.setStateText(6, 'Kalender 6');
C_5640_501_06_RTC01_KMD_MSV_R0544.setStateText(7, 'Kalender 7');
C_5640_501_06_RTC01_KMD_MSV_R0544.setStateText(8, 'Kalender 8');
C_5640_501_06_RTC01_KMD_MSV_R0544.setStateText(9, 'Kalender 9');
C_5640_501_06_RTC01_KMD_MSV_R0544.setStateText(10, 'Kalender 10');
A_360_01_SQ4_A407_KMD.setStateText(1, 'Auto');
A_360_01_SQ4_A407_KMD.setStateText(2, 'Åpne');
A_360_01_SQ4_A407_KMD.setStateText(3, 'Lukke');
A_360_01_SQ4_A407_KMD.setStateText(4, 'Til minste luftmengde');
A_360_01_SQ4_A407_KMD.setStateText(5, 'Til midterste luftmengde');
A_360_01_SQ4_A407_KMD.setStateText(6, 'Til største luftmengde');
A_360_01_SQ4_A407_KMD.setStateText(7, 'Åpne (rask)');
A_360_01_SQ4_A407_KMD.setStateText(8, 'Lukke (rask)');
A_360_01_SQ4_4AH2_KMD.setStateText(1, 'Auto');
A_360_01_SQ4_4AH2_KMD.setStateText(2, 'Åpne');
A_360_01_SQ4_4AH2_KMD.setStateText(3, 'Lukke');
A_360_01_SQ4_4AH2_KMD.setStateText(4, 'Til minste luftmengde');
A_360_01_SQ4_4AH2_KMD.setStateText(5, 'Til midterste luftmengde');
A_360_01_SQ4_4AH2_KMD.setStateText(6, 'Til største luftmengde');
A_360_01_SQ4_4AH2_KMD.setStateText(7, 'Åpne (rask)');
A_360_01_SQ4_4AH2_KMD.setStateText(8, 'Lukke (rask)');
A_360_01_SQ4_4AH1_KMD.setStateText(1, 'Auto');
A_360_01_SQ4_4AH1_KMD.setStateText(2, 'Åpne');
A_360_01_SQ4_4AH1_KMD.setStateText(3, 'Lukke');
A_360_01_SQ4_4AH1_KMD.setStateText(4, 'Til minste luftmengde');
A_360_01_SQ4_4AH1_KMD.setStateText(5, 'Til midterste luftmengde');
A_360_01_SQ4_4AH1_KMD.setStateText(6, 'Til største luftmengde');
A_360_01_SQ4_4AH1_KMD.setStateText(7, 'Åpne (rask)');
A_360_01_SQ4_4AH1_KMD.setStateText(8, 'Lukke (rask)');
A_360_01_SQ5_4AH1_KMD.setStateText(1, 'Auto');
A_360_01_SQ5_4AH1_KMD.setStateText(2, 'Åpne');
A_360_01_SQ5_4AH1_KMD.setStateText(3, 'Lukke');
A_360_01_SQ5_4AH1_KMD.setStateText(4, 'Til minste luftmengde');
A_360_01_SQ5_4AH1_KMD.setStateText(5, 'Til midterste luftmengde');
A_360_01_SQ5_4AH1_KMD.setStateText(6, 'Til største luftmengde');
A_360_01_SQ5_4AH1_KMD.setStateText(7, 'Åpne (rask)');
A_360_01_SQ5_4AH1_KMD.setStateText(8, 'Lukke (rask)');
A_360_01_SQ5_A405_KMD.setStateText(1, 'Auto');
A_360_01_SQ5_A405_KMD.setStateText(2, 'Åpne');
A_360_01_SQ5_A405_KMD.setStateText(3, 'Lukke');
A_360_01_SQ5_A405_KMD.setStateText(4, 'Til minste luftmengde');
A_360_01_SQ5_A405_KMD.setStateText(5, 'Til midterste luftmengde');
A_360_01_SQ5_A405_KMD.setStateText(6, 'Til største luftmengde');
A_360_01_SQ5_A405_KMD.setStateText(7, 'Åpne (rask)');
A_360_01_SQ5_A405_KMD.setStateText(8, 'Lukke (rask)');
A_360_01_SQ4_A401_2_KMD.setStateText(1, 'Auto');
A_360_01_SQ4_A401_2_KMD.setStateText(2, 'Åpne');
A_360_01_SQ4_A401_2_KMD.setStateText(3, 'Lukke');
A_360_01_SQ4_A401_2_KMD.setStateText(4, 'Til minste luftmengde');
A_360_01_SQ4_A401_2_KMD.setStateText(5, 'Til midterste luftmengde');
A_360_01_SQ4_A401_2_KMD.setStateText(6, 'Til største luftmengde');
A_360_01_SQ4_A401_2_KMD.setStateText(7, 'Åpne (rask)');
A_360_01_SQ4_A401_2_KMD.setStateText(8, 'Lukke (rask)');
A_360_01_SQ4_A401_1_KMD.setStateText(1, 'Auto');
A_360_01_SQ4_A401_1_KMD.setStateText(2, 'Åpne');
A_360_01_SQ4_A401_1_KMD.setStateText(3, 'Lukke');
A_360_01_SQ4_A401_1_KMD.setStateText(4, 'Til minste luftmengde');
A_360_01_SQ4_A401_1_KMD.setStateText(5, 'Til midterste luftmengde');
A_360_01_SQ4_A401_1_KMD.setStateText(6, 'Til største luftmengde');
A_360_01_SQ4_A401_1_KMD.setStateText(7, 'Åpne (rask)');
A_360_01_SQ4_A401_1_KMD.setStateText(8, 'Lukke (rask)');
A_360_01_SQ4_A401_KMD.setStateText(1, 'Auto');
A_360_01_SQ4_A401_KMD.setStateText(2, 'Åpne');
A_360_01_SQ4_A401_KMD.setStateText(3, 'Lukke');
A_360_01_SQ4_A401_KMD.setStateText(4, 'Til minste luftmengde');
A_360_01_SQ4_A401_KMD.setStateText(5, 'Til midterste luftmengde');
A_360_01_SQ4_A401_KMD.setStateText(6, 'Til største luftmengde');
A_360_01_SQ4_A401_KMD.setStateText(7, 'Åpne (rask)');
A_360_01_SQ4_A401_KMD.setStateText(8, 'Lukke (rask)');
A_360_01_SQ4_A406_KMD.setStateText(1, 'Auto');
A_360_01_SQ4_A406_KMD.setStateText(2, 'Åpne');
A_360_01_SQ4_A406_KMD.setStateText(3, 'Lukke');
A_360_01_SQ4_A406_KMD.setStateText(4, 'Til minste luftmengde');
A_360_01_SQ4_A406_KMD.setStateText(5, 'Til midterste luftmengde');
A_360_01_SQ4_A406_KMD.setStateText(6, 'Til største luftmengde');
A_360_01_SQ4_A406_KMD.setStateText(7, 'Åpne (rask)');
A_360_01_SQ4_A406_KMD.setStateText(8, 'Lukke (rask)');
A_360_01_SQ4_A408_KMD.setStateText(1, 'Auto');
A_360_01_SQ4_A408_KMD.setStateText(2, 'Åpne');
A_360_01_SQ4_A408_KMD.setStateText(3, 'Lukke');
A_360_01_SQ4_A408_KMD.setStateText(4, 'Til minste luftmengde');
A_360_01_SQ4_A408_KMD.setStateText(5, 'Til midterste luftmengde');
A_360_01_SQ4_A408_KMD.setStateText(6, 'Til største luftmengde');
A_360_01_SQ4_A408_KMD.setStateText(7, 'Åpne (rask)');
A_360_01_SQ4_A408_KMD.setStateText(8, 'Lukke (rask)');
A_360_01_SQ4_A410_1_KMD.setStateText(1, 'Auto');
A_360_01_SQ4_A410_1_KMD.setStateText(2, 'Åpne');
A_360_01_SQ4_A410_1_KMD.setStateText(3, 'Lukke');
A_360_01_SQ4_A410_1_KMD.setStateText(4, 'Til minste luftmengde');
A_360_01_SQ4_A410_1_KMD.setStateText(5, 'Til midterste luftmengde');
A_360_01_SQ4_A410_1_KMD.setStateText(6, 'Til største luftmengde');
A_360_01_SQ4_A410_1_KMD.setStateText(7, 'Åpne (rask)');
A_360_01_SQ4_A410_1_KMD.setStateText(8, 'Lukke (rask)');
A_360_01_SQ4_A410_2_KMD.setStateText(1, 'Auto');
A_360_01_SQ4_A410_2_KMD.setStateText(2, 'Åpne');
A_360_01_SQ4_A410_2_KMD.setStateText(3, 'Lukke');
A_360_01_SQ4_A410_2_KMD.setStateText(4, 'Til minste luftmengde');
A_360_01_SQ4_A410_2_KMD.setStateText(5, 'Til midterste luftmengde');
A_360_01_SQ4_A410_2_KMD.setStateText(6, 'Til største luftmengde');
A_360_01_SQ4_A410_2_KMD.setStateText(7, 'Åpne (rask)');
A_360_01_SQ4_A410_2_KMD.setStateText(8, 'Lukke (rask)');
A_360_01_SQ4_A410_3_KMD.setStateText(1, 'Auto');
A_360_01_SQ4_A410_3_KMD.setStateText(2, 'Åpne');
A_360_01_SQ4_A410_3_KMD.setStateText(3, 'Lukke');
A_360_01_SQ4_A410_3_KMD.setStateText(4, 'Til minste luftmengde');
A_360_01_SQ4_A410_3_KMD.setStateText(5, 'Til midterste luftmengde');
A_360_01_SQ4_A410_3_KMD.setStateText(6, 'Til største luftmengde');
A_360_01_SQ4_A410_3_KMD.setStateText(7, 'Åpne (rask)');
A_360_01_SQ4_A410_3_KMD.setStateText(8, 'Lukke (rask)');
A_360_01_SQ4_A410_4_KMD.setStateText(1, 'Auto');
A_360_01_SQ4_A410_4_KMD.setStateText(2, 'Åpne');
A_360_01_SQ4_A410_4_KMD.setStateText(3, 'Lukke');
A_360_01_SQ4_A410_4_KMD.setStateText(4, 'Til minste luftmengde');
A_360_01_SQ4_A410_4_KMD.setStateText(5, 'Til midterste luftmengde');
A_360_01_SQ4_A410_4_KMD.setStateText(6, 'Til største luftmengde');
A_360_01_SQ4_A410_4_KMD.setStateText(7, 'Åpne (rask)');
A_360_01_SQ4_A410_4_KMD.setStateText(8, 'Lukke (rask)');
A_360_01_SQ4_A410_5_KMD.setStateText(1, 'Auto');
A_360_01_SQ4_A410_5_KMD.setStateText(2, 'Åpne');
A_360_01_SQ4_A410_5_KMD.setStateText(3, 'Lukke');
A_360_01_SQ4_A410_5_KMD.setStateText(4, 'Til minste luftmengde');
A_360_01_SQ4_A410_5_KMD.setStateText(5, 'Til midterste luftmengde');
A_360_01_SQ4_A410_5_KMD.setStateText(6, 'Til største luftmengde');
A_360_01_SQ4_A410_5_KMD.setStateText(7, 'Åpne (rask)');
A_360_01_SQ4_A410_5_KMD.setStateText(8, 'Lukke (rask)');
A_360_01_SQ4_A412_KMD.setStateText(1, 'Auto');
A_360_01_SQ4_A412_KMD.setStateText(2, 'Åpne');
A_360_01_SQ4_A412_KMD.setStateText(3, 'Lukke');
A_360_01_SQ4_A412_KMD.setStateText(4, 'Til minste luftmengde');
A_360_01_SQ4_A412_KMD.setStateText(5, 'Til midterste luftmengde');
A_360_01_SQ4_A412_KMD.setStateText(6, 'Til største luftmengde');
A_360_01_SQ4_A412_KMD.setStateText(7, 'Åpne (rask)');
A_360_01_SQ4_A412_KMD.setStateText(8, 'Lukke (rask)');
A_360_01_SQ4_A413_KMD.setStateText(1, 'Auto');
A_360_01_SQ4_A413_KMD.setStateText(2, 'Åpne');
A_360_01_SQ4_A413_KMD.setStateText(3, 'Lukke');
A_360_01_SQ4_A413_KMD.setStateText(4, 'Til minste luftmengde');
A_360_01_SQ4_A413_KMD.setStateText(5, 'Til midterste luftmengde');
A_360_01_SQ4_A413_KMD.setStateText(6, 'Til største luftmengde');
A_360_01_SQ4_A413_KMD.setStateText(7, 'Åpne (rask)');
A_360_01_SQ4_A413_KMD.setStateText(8, 'Lukke (rask)');
A_360_01_SK4_A415_KMD.setStateText(1, 'Auto');
A_360_01_SK4_A415_KMD.setStateText(2, 'Åpne');
A_360_01_SK4_A415_KMD.setStateText(3, 'Lukke');
A_360_01_SK4_A415_KMD.setStateText(4, 'Til minste luftmengde');
A_360_01_SK4_A415_KMD.setStateText(5, 'Til midterste luftmengde');
A_360_01_SK4_A415_KMD.setStateText(6, 'Til største luftmengde');
A_360_01_SK4_A415_KMD.setStateText(7, 'Åpne (rask)');
A_360_01_SK4_A415_KMD.setStateText(8, 'Lukke (rask)');
A_360_01_SK5_A415_KMD.setStateText(1, 'Auto');
A_360_01_SK5_A415_KMD.setStateText(2, 'Åpne');
A_360_01_SK5_A415_KMD.setStateText(3, 'Lukke');
A_360_01_SK5_A415_KMD.setStateText(4, 'Til minste luftmengde');
A_360_01_SK5_A415_KMD.setStateText(5, 'Til midterste luftmengde');
A_360_01_SK5_A415_KMD.setStateText(6, 'Til største luftmengde');
A_360_01_SK5_A415_KMD.setStateText(7, 'Åpne (rask)');
A_360_01_SK5_A415_KMD.setStateText(8, 'Lukke (rask)');
A_360_01_SK5_A418_KMD.setStateText(1, 'Auto');
A_360_01_SK5_A418_KMD.setStateText(2, 'Åpne');
A_360_01_SK5_A418_KMD.setStateText(3, 'Lukke');
A_360_01_SK5_A418_KMD.setStateText(4, 'Til minste luftmengde');
A_360_01_SK5_A418_KMD.setStateText(5, 'Til midterste luftmengde');
A_360_01_SK5_A418_KMD.setStateText(6, 'Til største luftmengde');
A_360_01_SK5_A418_KMD.setStateText(7, 'Åpne (rask)');
A_360_01_SK5_A418_KMD.setStateText(8, 'Lukke (rask)');
A_360_01_SK4_A417_KMD.setStateText(1, 'Auto');
A_360_01_SK4_A417_KMD.setStateText(2, 'Åpne');
A_360_01_SK4_A417_KMD.setStateText(3, 'Lukke');
A_360_01_SK4_A417_KMD.setStateText(4, 'Til minste luftmengde');
A_360_01_SK4_A417_KMD.setStateText(5, 'Til midterste luftmengde');
A_360_01_SK4_A417_KMD.setStateText(6, 'Til største luftmengde');
A_360_01_SK4_A417_KMD.setStateText(7, 'Åpne (rask)');
A_360_01_SK4_A417_KMD.setStateText(8, 'Lukke (rask)');
A_360_01_SQ5_C411_KMD.setStateText(1, 'Auto');
A_360_01_SQ5_C411_KMD.setStateText(2, 'Åpne');
A_360_01_SQ5_C411_KMD.setStateText(3, 'Lukke');
A_360_01_SQ5_C411_KMD.setStateText(4, 'Til minste luftmengde');
A_360_01_SQ5_C411_KMD.setStateText(5, 'Til midterste luftmengde');
A_360_01_SQ5_C411_KMD.setStateText(6, 'Til største luftmengde');
A_360_01_SQ5_C411_KMD.setStateText(7, 'Åpne (rask)');
A_360_01_SQ5_C411_KMD.setStateText(8, 'Lukke (rask)');
A_360_01_SK5_A421_KMD.setStateText(1, 'Auto');
A_360_01_SK5_A421_KMD.setStateText(2, 'Åpne');
A_360_01_SK5_A421_KMD.setStateText(3, 'Lukke');
A_360_01_SK5_A421_KMD.setStateText(4, 'Til minste luftmengde');
A_360_01_SK5_A421_KMD.setStateText(5, 'Til midterste luftmengde');
A_360_01_SK5_A421_KMD.setStateText(6, 'Til største luftmengde');
A_360_01_SK5_A421_KMD.setStateText(7, 'Åpne (rask)');
A_360_01_SK5_A421_KMD.setStateText(8, 'Lukke (rask)');
A_360_01_SQ5_4AH2_KMD.setStateText(1, 'Auto');
A_360_01_SQ5_4AH2_KMD.setStateText(2, 'Åpne');
A_360_01_SQ5_4AH2_KMD.setStateText(3, 'Lukke');
A_360_01_SQ5_4AH2_KMD.setStateText(4, 'Til minste luftmengde');
A_360_01_SQ5_4AH2_KMD.setStateText(5, 'Til midterste luftmengde');
A_360_01_SQ5_4AH2_KMD.setStateText(6, 'Til største luftmengde');
A_360_01_SQ5_4AH2_KMD.setStateText(7, 'Åpne (rask)');
A_360_01_SQ5_4AH2_KMD.setStateText(8, 'Lukke (rask)');
A_360_01_SK5_A424_KMD.setStateText(1, 'Auto');
A_360_01_SK5_A424_KMD.setStateText(2, 'Åpne');
A_360_01_SK5_A424_KMD.setStateText(3, 'Lukke');
A_360_01_SK5_A424_KMD.setStateText(4, 'Til minste luftmengde');
A_360_01_SK5_A424_KMD.setStateText(5, 'Til midterste luftmengde');
A_360_01_SK5_A424_KMD.setStateText(6, 'Til største luftmengde');
A_360_01_SK5_A424_KMD.setStateText(7, 'Åpne (rask)');
A_360_01_SK5_A424_KMD.setStateText(8, 'Lukke (rask)');
A_360_01_SQ4_4AH3_KMD.setStateText(1, 'Auto');
A_360_01_SQ4_4AH3_KMD.setStateText(2, 'Åpne');
A_360_01_SQ4_4AH3_KMD.setStateText(3, 'Lukke');
A_360_01_SQ4_4AH3_KMD.setStateText(4, 'Til minste luftmengde');
A_360_01_SQ4_4AH3_KMD.setStateText(5, 'Til midterste luftmengde');
A_360_01_SQ4_4AH3_KMD.setStateText(6, 'Til største luftmengde');
A_360_01_SQ4_4AH3_KMD.setStateText(7, 'Åpne (rask)');
A_360_01_SQ4_4AH3_KMD.setStateText(8, 'Lukke (rask)');
A_360_01_SQ4_4AH4_KMD.setStateText(1, 'Auto');
A_360_01_SQ4_4AH4_KMD.setStateText(2, 'Åpne');
A_360_01_SQ4_4AH4_KMD.setStateText(3, 'Lukke');
A_360_01_SQ4_4AH4_KMD.setStateText(4, 'Til minste luftmengde');
A_360_01_SQ4_4AH4_KMD.setStateText(5, 'Til midterste luftmengde');
A_360_01_SQ4_4AH4_KMD.setStateText(6, 'Til største luftmengde');
A_360_01_SQ4_4AH4_KMD.setStateText(7, 'Åpne (rask)');
A_360_01_SQ4_4AH4_KMD.setStateText(8, 'Lukke (rask)');
A_360_01_SQ4_4AH5_KMD.setStateText(1, 'Auto');
A_360_01_SQ4_4AH5_KMD.setStateText(2, 'Åpne');
A_360_01_SQ4_4AH5_KMD.setStateText(3, 'Lukke');
A_360_01_SQ4_4AH5_KMD.setStateText(4, 'Til minste luftmengde');
A_360_01_SQ4_4AH5_KMD.setStateText(5, 'Til midterste luftmengde');
A_360_01_SQ4_4AH5_KMD.setStateText(6, 'Til største luftmengde');
A_360_01_SQ4_4AH5_KMD.setStateText(7, 'Åpne (rask)');
A_360_01_SQ4_4AH5_KMD.setStateText(8, 'Lukke (rask)');
A_360_01_SQ5_4AH3_KMD.setStateText(1, 'Auto');
A_360_01_SQ5_4AH3_KMD.setStateText(2, 'Åpne');
A_360_01_SQ5_4AH3_KMD.setStateText(3, 'Lukke');
A_360_01_SQ5_4AH3_KMD.setStateText(4, 'Til minste luftmengde');
A_360_01_SQ5_4AH3_KMD.setStateText(5, 'Til midterste luftmengde');
A_360_01_SQ5_4AH3_KMD.setStateText(6, 'Til største luftmengde');
A_360_01_SQ5_4AH3_KMD.setStateText(7, 'Åpne (rask)');
A_360_01_SQ5_4AH3_KMD.setStateText(8, 'Lukke (rask)');
A_360_01_SQ5_A401_KMD.setStateText(1, 'Auto');
A_360_01_SQ5_A401_KMD.setStateText(2, 'Åpne');
A_360_01_SQ5_A401_KMD.setStateText(3, 'Lukke');
A_360_01_SQ5_A401_KMD.setStateText(4, 'Til minste luftmengde');
A_360_01_SQ5_A401_KMD.setStateText(5, 'Til midterste luftmengde');
A_360_01_SQ5_A401_KMD.setStateText(6, 'Til største luftmengde');
A_360_01_SQ5_A401_KMD.setStateText(7, 'Åpne (rask)');
A_360_01_SQ5_A401_KMD.setStateText(8, 'Lukke (rask)');
A_360_01_SQ4_A403_KMD.setStateText(1, 'Auto');
A_360_01_SQ4_A403_KMD.setStateText(2, 'Åpne');
A_360_01_SQ4_A403_KMD.setStateText(3, 'Lukke');
A_360_01_SQ4_A403_KMD.setStateText(4, 'Til minste luftmengde');
A_360_01_SQ4_A403_KMD.setStateText(5, 'Til midterste luftmengde');
A_360_01_SQ4_A403_KMD.setStateText(6, 'Til største luftmengde');
A_360_01_SQ4_A403_KMD.setStateText(7, 'Åpne (rask)');
A_360_01_SQ4_A403_KMD.setStateText(8, 'Lukke (rask)');
A_360_01_SQ4_A401_3_KMD.setStateText(1, 'Auto');
A_360_01_SQ4_A401_3_KMD.setStateText(2, 'Åpne');
A_360_01_SQ4_A401_3_KMD.setStateText(3, 'Lukke');
A_360_01_SQ4_A401_3_KMD.setStateText(4, 'Til minste luftmengde');
A_360_01_SQ4_A401_3_KMD.setStateText(5, 'Til midterste luftmengde');
A_360_01_SQ4_A401_3_KMD.setStateText(6, 'Til største luftmengde');
A_360_01_SQ4_A401_3_KMD.setStateText(7, 'Åpne (rask)');
A_360_01_SQ4_A401_3_KMD.setStateText(8, 'Lukke (rask)');
A_360_01_SQ4_A401_4_KMD.setStateText(1, 'Auto');
A_360_01_SQ4_A401_4_KMD.setStateText(2, 'Åpne');
A_360_01_SQ4_A401_4_KMD.setStateText(3, 'Lukke');
A_360_01_SQ4_A401_4_KMD.setStateText(4, 'Til minste luftmengde');
A_360_01_SQ4_A401_4_KMD.setStateText(5, 'Til midterste luftmengde');
A_360_01_SQ4_A401_4_KMD.setStateText(6, 'Til største luftmengde');
A_360_01_SQ4_A401_4_KMD.setStateText(7, 'Åpne (rask)');
A_360_01_SQ4_A401_4_KMD.setStateText(8, 'Lukke (rask)');
A_360_01_SQ4_A401_5_KMD.setStateText(1, 'Auto');
A_360_01_SQ4_A401_5_KMD.setStateText(2, 'Åpne');
A_360_01_SQ4_A401_5_KMD.setStateText(3, 'Lukke');
A_360_01_SQ4_A401_5_KMD.setStateText(4, 'Til minste luftmengde');
A_360_01_SQ4_A401_5_KMD.setStateText(5, 'Til midterste luftmengde');
A_360_01_SQ4_A401_5_KMD.setStateText(6, 'Til største luftmengde');
A_360_01_SQ4_A401_5_KMD.setStateText(7, 'Åpne (rask)');
A_360_01_SQ4_A401_5_KMD.setStateText(8, 'Lukke (rask)');
A_360_01_SQ4_A401_6_KMD.setStateText(1, 'Auto');
A_360_01_SQ4_A401_6_KMD.setStateText(2, 'Åpne');
A_360_01_SQ4_A401_6_KMD.setStateText(3, 'Lukke');
A_360_01_SQ4_A401_6_KMD.setStateText(4, 'Til minste luftmengde');
A_360_01_SQ4_A401_6_KMD.setStateText(5, 'Til midterste luftmengde');
A_360_01_SQ4_A401_6_KMD.setStateText(6, 'Til største luftmengde');
A_360_01_SQ4_A401_6_KMD.setStateText(7, 'Åpne (rask)');
A_360_01_SQ4_A401_6_KMD.setStateText(8, 'Lukke (rask)');
A_360_01_SQ4_A401_7_KMD.setStateText(1, 'Auto');
A_360_01_SQ4_A401_7_KMD.setStateText(2, 'Åpne');
A_360_01_SQ4_A401_7_KMD.setStateText(3, 'Lukke');
A_360_01_SQ4_A401_7_KMD.setStateText(4, 'Til minste luftmengde');
A_360_01_SQ4_A401_7_KMD.setStateText(5, 'Til midterste luftmengde');
A_360_01_SQ4_A401_7_KMD.setStateText(6, 'Til største luftmengde');
A_360_01_SQ4_A401_7_KMD.setStateText(7, 'Åpne (rask)');
A_360_01_SQ4_A401_7_KMD.setStateText(8, 'Lukke (rask)');
A_360_01_SQ4_A401_8_KMD.setStateText(1, 'Auto');
A_360_01_SQ4_A401_8_KMD.setStateText(2, 'Åpne');
A_360_01_SQ4_A401_8_KMD.setStateText(3, 'Lukke');
A_360_01_SQ4_A401_8_KMD.setStateText(4, 'Til minste luftmengde');
A_360_01_SQ4_A401_8_KMD.setStateText(5, 'Til midterste luftmengde');
A_360_01_SQ4_A401_8_KMD.setStateText(6, 'Til største luftmengde');
A_360_01_SQ4_A401_8_KMD.setStateText(7, 'Åpne (rask)');
A_360_01_SQ4_A401_8_KMD.setStateText(8, 'Lukke (rask)');
A_360_01_SQ4_A401_9_KMD.setStateText(1, 'Auto');
A_360_01_SQ4_A401_9_KMD.setStateText(2, 'Åpne');
A_360_01_SQ4_A401_9_KMD.setStateText(3, 'Lukke');
A_360_01_SQ4_A401_9_KMD.setStateText(4, 'Til minste luftmengde');
A_360_01_SQ4_A401_9_KMD.setStateText(5, 'Til midterste luftmengde');
A_360_01_SQ4_A401_9_KMD.setStateText(6, 'Til største luftmengde');
A_360_01_SQ4_A401_9_KMD.setStateText(7, 'Åpne (rask)');
A_360_01_SQ4_A401_9_KMD.setStateText(8, 'Lukke (rask)');
A_360_01_SQ4_A401_0_KMD.setStateText(1, 'Auto');
A_360_01_SQ4_A401_0_KMD.setStateText(2, 'Åpne');
A_360_01_SQ4_A401_0_KMD.setStateText(3, 'Lukke');
A_360_01_SQ4_A401_0_KMD.setStateText(4, 'Til minste luftmengde');
A_360_01_SQ4_A401_0_KMD.setStateText(5, 'Til midterste luftmengde');
A_360_01_SQ4_A401_0_KMD.setStateText(6, 'Til største luftmengde');
A_360_01_SQ4_A401_0_KMD.setStateText(7, 'Åpne (rask)');
A_360_01_SQ4_A401_0_KMD.setStateText(8, 'Lukke (rask)');
A_360_01_SQ4_A426_KMD.setStateText(1, 'Auto');
A_360_01_SQ4_A426_KMD.setStateText(2, 'Åpne');
A_360_01_SQ4_A426_KMD.setStateText(3, 'Lukke');
A_360_01_SQ4_A426_KMD.setStateText(4, 'Til minste luftmengde');
A_360_01_SQ4_A426_KMD.setStateText(5, 'Til midterste luftmengde');
A_360_01_SQ4_A426_KMD.setStateText(6, 'Til største luftmengde');
A_360_01_SQ4_A426_KMD.setStateText(7, 'Åpne (rask)');
A_360_01_SQ4_A426_KMD.setStateText(8, 'Lukke (rask)');
A_360_01_SQ4_A428_1_KMD.setStateText(1, 'Auto');
A_360_01_SQ4_A428_1_KMD.setStateText(2, 'Åpne');
A_360_01_SQ4_A428_1_KMD.setStateText(3, 'Lukke');
A_360_01_SQ4_A428_1_KMD.setStateText(4, 'Til minste luftmengde');
A_360_01_SQ4_A428_1_KMD.setStateText(5, 'Til midterste luftmengde');
A_360_01_SQ4_A428_1_KMD.setStateText(6, 'Til største luftmengde');
A_360_01_SQ4_A428_1_KMD.setStateText(7, 'Åpne (rask)');
A_360_01_SQ4_A428_1_KMD.setStateText(8, 'Lukke (rask)');
A_360_01_SQ4_A428_2_KMD.setStateText(1, 'Auto');
A_360_01_SQ4_A428_2_KMD.setStateText(2, 'Åpne');
A_360_01_SQ4_A428_2_KMD.setStateText(3, 'Lukke');
A_360_01_SQ4_A428_2_KMD.setStateText(4, 'Til minste luftmengde');
A_360_01_SQ4_A428_2_KMD.setStateText(5, 'Til midterste luftmengde');
A_360_01_SQ4_A428_2_KMD.setStateText(6, 'Til største luftmengde');
A_360_01_SQ4_A428_2_KMD.setStateText(7, 'Åpne (rask)');
A_360_01_SQ4_A428_2_KMD.setStateText(8, 'Lukke (rask)');
A_360_01_SQ4_A428_3_KMD.setStateText(1, 'Auto');
A_360_01_SQ4_A428_3_KMD.setStateText(2, 'Åpne');
A_360_01_SQ4_A428_3_KMD.setStateText(3, 'Lukke');
A_360_01_SQ4_A428_3_KMD.setStateText(4, 'Til minste luftmengde');
A_360_01_SQ4_A428_3_KMD.setStateText(5, 'Til midterste luftmengde');
A_360_01_SQ4_A428_3_KMD.setStateText(6, 'Til største luftmengde');
A_360_01_SQ4_A428_3_KMD.setStateText(7, 'Åpne (rask)');
A_360_01_SQ4_A428_3_KMD.setStateText(8, 'Lukke (rask)');
A_360_01_SQ4_A428_4_KMD.setStateText(1, 'Auto');
A_360_01_SQ4_A428_4_KMD.setStateText(2, 'Åpne');
A_360_01_SQ4_A428_4_KMD.setStateText(3, 'Lukke');
A_360_01_SQ4_A428_4_KMD.setStateText(4, 'Til minste luftmengde');
A_360_01_SQ4_A428_4_KMD.setStateText(5, 'Til midterste luftmengde');
A_360_01_SQ4_A428_4_KMD.setStateText(6, 'Til største luftmengde');
A_360_01_SQ4_A428_4_KMD.setStateText(7, 'Åpne (rask)');
A_360_01_SQ4_A428_4_KMD.setStateText(8, 'Lukke (rask)');
A_360_01_SQ5_A425_KMD.setStateText(1, 'Auto');
A_360_01_SQ5_A425_KMD.setStateText(2, 'Åpne');
A_360_01_SQ5_A425_KMD.setStateText(3, 'Lukke');
A_360_01_SQ5_A425_KMD.setStateText(4, 'Til minste luftmengde');
A_360_01_SQ5_A425_KMD.setStateText(5, 'Til midterste luftmengde');
A_360_01_SQ5_A425_KMD.setStateText(6, 'Til største luftmengde');
A_360_01_SQ5_A425_KMD.setStateText(7, 'Åpne (rask)');
A_360_01_SQ5_A425_KMD.setStateText(8, 'Lukke (rask)');
A_360_01_SQ4_A428_5_KMD.setStateText(1, 'Auto');
A_360_01_SQ4_A428_5_KMD.setStateText(2, 'Åpne');
A_360_01_SQ4_A428_5_KMD.setStateText(3, 'Lukke');
A_360_01_SQ4_A428_5_KMD.setStateText(4, 'Til minste luftmengde');
A_360_01_SQ4_A428_5_KMD.setStateText(5, 'Til midterste luftmengde');
A_360_01_SQ4_A428_5_KMD.setStateText(6, 'Til største luftmengde');
A_360_01_SQ4_A428_5_KMD.setStateText(7, 'Åpne (rask)');
A_360_01_SQ4_A428_5_KMD.setStateText(8, 'Lukke (rask)');
A_360_01_SQ4_A428_6_KMD.setStateText(1, 'Auto');
A_360_01_SQ4_A428_6_KMD.setStateText(2, 'Åpne');
A_360_01_SQ4_A428_6_KMD.setStateText(3, 'Lukke');
A_360_01_SQ4_A428_6_KMD.setStateText(4, 'Til minste luftmengde');
A_360_01_SQ4_A428_6_KMD.setStateText(5, 'Til midterste luftmengde');
A_360_01_SQ4_A428_6_KMD.setStateText(6, 'Til største luftmengde');
A_360_01_SQ4_A428_6_KMD.setStateText(7, 'Åpne (rask)');
A_360_01_SQ4_A428_6_KMD.setStateText(8, 'Lukke (rask)');
A_360_01_SQ4_A428_7_KMD.setStateText(1, 'Auto');
A_360_01_SQ4_A428_7_KMD.setStateText(2, 'Åpne');
A_360_01_SQ4_A428_7_KMD.setStateText(3, 'Lukke');
A_360_01_SQ4_A428_7_KMD.setStateText(4, 'Til minste luftmengde');
A_360_01_SQ4_A428_7_KMD.setStateText(5, 'Til midterste luftmengde');
A_360_01_SQ4_A428_7_KMD.setStateText(6, 'Til største luftmengde');
A_360_01_SQ4_A428_7_KMD.setStateText(7, 'Åpne (rask)');
A_360_01_SQ4_A428_7_KMD.setStateText(8, 'Lukke (rask)');
B_360_02_SQ5_UBH1_KMD.setStateText(1, 'Auto');
B_360_02_SQ5_UBH1_KMD.setStateText(2, 'Åpne');
B_360_02_SQ5_UBH1_KMD.setStateText(3, 'Lukke');
B_360_02_SQ5_UBH1_KMD.setStateText(4, 'Til minste luftmengde');
B_360_02_SQ5_UBH1_KMD.setStateText(5, 'Til midterste luftmengde');
B_360_02_SQ5_UBH1_KMD.setStateText(6, 'Til største luftmengde');
B_360_02_SQ5_UBH1_KMD.setStateText(7, 'Åpne (rask)');
B_360_02_SQ5_UBH1_KMD.setStateText(8, 'Lukke (rask)');
B_360_02_SQ5_UBH2_KMD.setStateText(1, 'Auto');
B_360_02_SQ5_UBH2_KMD.setStateText(2, 'Åpne');
B_360_02_SQ5_UBH2_KMD.setStateText(3, 'Lukke');
B_360_02_SQ5_UBH2_KMD.setStateText(4, 'Til minste luftmengde');
B_360_02_SQ5_UBH2_KMD.setStateText(5, 'Til midterste luftmengde');
B_360_02_SQ5_UBH2_KMD.setStateText(6, 'Til største luftmengde');
B_360_02_SQ5_UBH2_KMD.setStateText(7, 'Åpne (rask)');
B_360_02_SQ5_UBH2_KMD.setStateText(8, 'Lukke (rask)');
B_360_02_SQ4_UBH1_KMD.setStateText(1, 'Auto');
B_360_02_SQ4_UBH1_KMD.setStateText(2, 'Åpne');
B_360_02_SQ4_UBH1_KMD.setStateText(3, 'Lukke');
B_360_02_SQ4_UBH1_KMD.setStateText(4, 'Til minste luftmengde');
B_360_02_SQ4_UBH1_KMD.setStateText(5, 'Til midterste luftmengde');
B_360_02_SQ4_UBH1_KMD.setStateText(6, 'Til største luftmengde');
B_360_02_SQ4_UBH1_KMD.setStateText(7, 'Åpne (rask)');
B_360_02_SQ4_UBH1_KMD.setStateText(8, 'Lukke (rask)');
B_360_02_SQ4_UBH2_KMD.setStateText(1, 'Auto');
B_360_02_SQ4_UBH2_KMD.setStateText(2, 'Åpne');
B_360_02_SQ4_UBH2_KMD.setStateText(3, 'Lukke');
B_360_02_SQ4_UBH2_KMD.setStateText(4, 'Til minste luftmengde');
B_360_02_SQ4_UBH2_KMD.setStateText(5, 'Til midterste luftmengde');
B_360_02_SQ4_UBH2_KMD.setStateText(6, 'Til største luftmengde');
B_360_02_SQ4_UBH2_KMD.setStateText(7, 'Åpne (rask)');
B_360_02_SQ4_UBH2_KMD.setStateText(8, 'Lukke (rask)');
END_IF
                
              
END_PROGRAM

PROGRAM PRG_Mapping
  VAR
    bacnetModbusClimateInterop : ARRAY[0..22] OF bacnetModbusClimateInterop_00_01;
    bacnetModbusDamperInterop : ARRAY[1..GVL_Modbus.numberOfModbusDamperLines] OF ARRAY [1..30] OF bacnetModbusDamperInterop_00_01;
    i : INT;
  END_VAR

                
    i := 0;

                
// Mappinger for rom 401

bacnetModbusClimateInterop[i](
  BO_PresenceDetection			:= C_5640_501_06_RBA01_D_R0401,
  AI_CurrentTemperature			:= C_5640_501_06_RTC01_MV_R0401,
  AV_CurrentHeatingSetpoint		:= C_5640_501_06_RTC01_SPV_R0401,
  AV_ComfortHeatingSetpoint		:= C_5640_501_06_RTC01_SPV_Komf_R0401,
  AV_StandbyHeatingSetpoint		:= C_5640_501_06_RTC01_SPV_Stdb_R0401,
  AV_EconomyHeatingSetpoint		:= C_5640_501_06_RTC01_SPV_Natt_R0401,
  MSV_CurrentWorkingMode			:= C_5640_501_06_RTC01_MOD_FB_R0401,
  MSV_Calendar					:= C_5640_501_06_RTC01_KMD_MSV_R0401,
  AV_PresenceDelayOff				:= C_5640_501_06_RTC01_SP_Tid_Stdb_R0401,
  AV_SetpointAirQuality			:= C_5640_501_06_RYA601_SP_R0401,
  AI_CurrentCo2					:= C_5640_501_06_RYA601_MV_R0401,
  AO_ControlledVariableHeating	:= C_5640_501_06_SBB01_C_R0401,
  modbusHoldingRegisters		:= ADR(GVL_Modbus.awHoldingRegisters[i * 40]), 
  modbusCoilRegisters			:= ADR(GVL_Modbus.axCoils[i]), 
  typClimateControllerInterface	:= GVL_ClimateControl.typClimateControllerInterfaceRoom401, 
  typClimateControllerSettings  := PersistentVars.typClimateControllerSettingsRoom401
);
i := i +1;
                
// Mappinger for rom 406

bacnetModbusClimateInterop[i](
  BO_PresenceDetection			:= C_5640_501_06_RBA01_D_R0406,
  AI_CurrentTemperature			:= C_5640_501_06_RTC01_MV_R0406,
  AV_CurrentHeatingSetpoint		:= C_5640_501_06_RTC01_SPV_R0406,
  AV_ComfortHeatingSetpoint		:= C_5640_501_06_RTC01_SPV_Komf_R0406,
  AV_StandbyHeatingSetpoint		:= C_5640_501_06_RTC01_SPV_Stdb_R0406,
  AV_EconomyHeatingSetpoint		:= C_5640_501_06_RTC01_SPV_Natt_R0406,
  MSV_CurrentWorkingMode			:= C_5640_501_06_RTC01_MOD_FB_R0406,
  MSV_Calendar					:= C_5640_501_06_RTC01_KMD_MSV_R0406,
  AV_PresenceDelayOff				:= C_5640_501_06_RTC01_SP_Tid_Stdb_R0406,
  AV_SetpointAirQuality			:= C_5640_501_06_RYA601_SP_R0406,
  AI_CurrentCo2					:= C_5640_501_06_RYA601_MV_R0406,
  AO_ControlledVariableHeating	:= C_5640_501_06_SBB01_C_R0406,
  modbusHoldingRegisters		:= ADR(GVL_Modbus.awHoldingRegisters[i * 40]), 
  modbusCoilRegisters			:= ADR(GVL_Modbus.axCoils[i]), 
  typClimateControllerInterface	:= GVL_ClimateControl.typClimateControllerInterfaceRoom406, 
  typClimateControllerSettings  := PersistentVars.typClimateControllerSettingsRoom406
);
i := i +1;
                
// Mappinger for rom 407

bacnetModbusClimateInterop[i](
  BO_PresenceDetection			:= C_5640_501_06_RBA01_D_R0407,
  AI_CurrentTemperature			:= C_5640_501_06_RTC01_MV_R0407,
  AV_CurrentHeatingSetpoint		:= C_5640_501_06_RTC01_SPV_R0407,
  AV_ComfortHeatingSetpoint		:= C_5640_501_06_RTC01_SPV_Komf_R0407,
  AV_StandbyHeatingSetpoint		:= C_5640_501_06_RTC01_SPV_Stdb_R0407,
  AV_EconomyHeatingSetpoint		:= C_5640_501_06_RTC01_SPV_Natt_R0407,
  MSV_CurrentWorkingMode			:= C_5640_501_06_RTC01_MOD_FB_R0407,
  MSV_Calendar					:= C_5640_501_06_RTC01_KMD_MSV_R0407,
  AV_PresenceDelayOff				:= C_5640_501_06_RTC01_SP_Tid_Stdb_R0407,
  AV_SetpointAirQuality			:= C_5640_501_06_RYA601_SP_R0407,
  AI_CurrentCo2					:= C_5640_501_06_RYA601_MV_R0407,
  AO_ControlledVariableHeating	:= C_5640_501_06_SBB01_C_R0407,
  modbusHoldingRegisters		:= ADR(GVL_Modbus.awHoldingRegisters[i * 40]), 
  modbusCoilRegisters			:= ADR(GVL_Modbus.axCoils[i]), 
  typClimateControllerInterface	:= GVL_ClimateControl.typClimateControllerInterfaceRoom407, 
  typClimateControllerSettings  := PersistentVars.typClimateControllerSettingsRoom407
);
i := i +1;
                
// Mappinger for rom 408

bacnetModbusClimateInterop[i](
  BO_PresenceDetection			:= C_5640_501_06_RBA01_D_R0408,
  AI_CurrentTemperature			:= C_5640_501_06_RTC01_MV_R0408,
  AV_CurrentHeatingSetpoint		:= C_5640_501_06_RTC01_SPV_R0408,
  AV_ComfortHeatingSetpoint		:= C_5640_501_06_RTC01_SPV_Komf_R0408,
  AV_StandbyHeatingSetpoint		:= C_5640_501_06_RTC01_SPV_Stdb_R0408,
  AV_EconomyHeatingSetpoint		:= C_5640_501_06_RTC01_SPV_Natt_R0408,
  MSV_CurrentWorkingMode			:= C_5640_501_06_RTC01_MOD_FB_R0408,
  MSV_Calendar					:= C_5640_501_06_RTC01_KMD_MSV_R0408,
  AV_PresenceDelayOff				:= C_5640_501_06_RTC01_SP_Tid_Stdb_R0408,
  AV_SetpointAirQuality			:= C_5640_501_06_RYA601_SP_R0408,
  AI_CurrentCo2					:= C_5640_501_06_RYA601_MV_R0408,
  AO_ControlledVariableHeating	:= C_5640_501_06_SBB01_C_R0408,
  modbusHoldingRegisters		:= ADR(GVL_Modbus.awHoldingRegisters[i * 40]), 
  modbusCoilRegisters			:= ADR(GVL_Modbus.axCoils[i]), 
  typClimateControllerInterface	:= GVL_ClimateControl.typClimateControllerInterfaceRoom408, 
  typClimateControllerSettings  := PersistentVars.typClimateControllerSettingsRoom408
);
i := i +1;
                
// Mappinger for rom 409

bacnetModbusClimateInterop[i](
  BO_PresenceDetection			:= C_5640_501_06_RBA01_D_R0409,
  AI_CurrentTemperature			:= C_5640_501_06_RTC01_MV_R0409,
  AV_CurrentHeatingSetpoint		:= C_5640_501_06_RTC01_SPV_R0409,
  AV_ComfortHeatingSetpoint		:= C_5640_501_06_RTC01_SPV_Komf_R0409,
  AV_StandbyHeatingSetpoint		:= C_5640_501_06_RTC01_SPV_Stdb_R0409,
  AV_EconomyHeatingSetpoint		:= C_5640_501_06_RTC01_SPV_Natt_R0409,
  MSV_CurrentWorkingMode			:= C_5640_501_06_RTC01_MOD_FB_R0409,
  MSV_Calendar					:= C_5640_501_06_RTC01_KMD_MSV_R0409,
  AV_PresenceDelayOff				:= C_5640_501_06_RTC01_SP_Tid_Stdb_R0409,
  AV_SetpointAirQuality			:= C_5640_501_06_RYA601_SP_R0409,
  AI_CurrentCo2					:= C_5640_501_06_RYA601_MV_R0409,
  AO_ControlledVariableHeating	:= C_5640_501_06_SBB01_C_R0409,
  modbusHoldingRegisters		:= ADR(GVL_Modbus.awHoldingRegisters[i * 40]), 
  modbusCoilRegisters			:= ADR(GVL_Modbus.axCoils[i]), 
  typClimateControllerInterface	:= GVL_ClimateControl.typClimateControllerInterfaceRoom409, 
  typClimateControllerSettings  := PersistentVars.typClimateControllerSettingsRoom409
);
i := i +1;
                
// Mappinger for rom 464

bacnetModbusClimateInterop[i](
  BO_PresenceDetection			:= C_5640_501_06_RBA01_D_R0464,
  AI_CurrentTemperature			:= C_5640_501_06_RTC01_MV_R0464,
  AV_CurrentHeatingSetpoint		:= C_5640_501_06_RTC01_SPV_R0464,
  AV_ComfortHeatingSetpoint		:= C_5640_501_06_RTC01_SPV_Komf_R0464,
  AV_StandbyHeatingSetpoint		:= C_5640_501_06_RTC01_SPV_Stdb_R0464,
  AV_EconomyHeatingSetpoint		:= C_5640_501_06_RTC01_SPV_Natt_R0464,
  MSV_CurrentWorkingMode			:= C_5640_501_06_RTC01_MOD_FB_R0464,
  MSV_Calendar					:= C_5640_501_06_RTC01_KMD_MSV_R0464,
  AV_PresenceDelayOff				:= C_5640_501_06_RTC01_SP_Tid_Stdb_R0464,
  AV_SetpointAirQuality			:= C_5640_501_06_RYA601_SP_R0464,
  AI_CurrentCo2					:= C_5640_501_06_RYA601_MV_R0464,
  AO_ControlledVariableHeating	:= C_5640_501_06_SBB01_C_R0464,
  modbusHoldingRegisters		:= ADR(GVL_Modbus.awHoldingRegisters[i * 40]), 
  modbusCoilRegisters			:= ADR(GVL_Modbus.axCoils[i]), 
  typClimateControllerInterface	:= GVL_ClimateControl.typClimateControllerInterfaceRoom464, 
  typClimateControllerSettings  := PersistentVars.typClimateControllerSettingsRoom464
);
i := i +1;
                
// Mappinger for rom 415

bacnetModbusClimateInterop[i](
  BO_PresenceDetection			:= C_5640_501_06_RBA01_D_R0415,
  AI_CurrentTemperature			:= C_5640_501_06_RTC01_MV_R0415,
  AV_CurrentHeatingSetpoint		:= C_5640_501_06_RTC01_SPV_R0415,
  AV_ComfortHeatingSetpoint		:= C_5640_501_06_RTC01_SPV_Komf_R0415,
  AV_StandbyHeatingSetpoint		:= C_5640_501_06_RTC01_SPV_Stdb_R0415,
  AV_EconomyHeatingSetpoint		:= C_5640_501_06_RTC01_SPV_Natt_R0415,
  MSV_CurrentWorkingMode			:= C_5640_501_06_RTC01_MOD_FB_R0415,
  MSV_Calendar					:= C_5640_501_06_RTC01_KMD_MSV_R0415,
  AV_PresenceDelayOff				:= C_5640_501_06_RTC01_SP_Tid_Stdb_R0415,
  AV_SetpointAirQuality			:= C_5640_501_06_RYA601_SP_R0415,
  AI_CurrentCo2					:= C_5640_501_06_RYA601_MV_R0415,
  AO_ControlledVariableHeating	:= C_5640_501_06_SBB01_C_R0415,
  modbusHoldingRegisters		:= ADR(GVL_Modbus.awHoldingRegisters[i * 40]), 
  modbusCoilRegisters			:= ADR(GVL_Modbus.axCoils[i]), 
  typClimateControllerInterface	:= GVL_ClimateControl.typClimateControllerInterfaceRoom415, 
  typClimateControllerSettings  := PersistentVars.typClimateControllerSettingsRoom415
);
i := i +1;
                
// Mappinger for rom 422

bacnetModbusClimateInterop[i](
  BO_PresenceDetection			:= C_5640_501_06_RBA01_D_R0422,
  AI_CurrentTemperature			:= C_5640_501_06_RTC01_MV_R0422,
  AV_CurrentHeatingSetpoint		:= C_5640_501_06_RTC01_SPV_R0422,
  AV_ComfortHeatingSetpoint		:= C_5640_501_06_RTC01_SPV_Komf_R0422,
  AV_StandbyHeatingSetpoint		:= C_5640_501_06_RTC01_SPV_Stdb_R0422,
  AV_EconomyHeatingSetpoint		:= C_5640_501_06_RTC01_SPV_Natt_R0422,
  MSV_CurrentWorkingMode			:= C_5640_501_06_RTC01_MOD_FB_R0422,
  MSV_Calendar					:= C_5640_501_06_RTC01_KMD_MSV_R0422,
  AV_PresenceDelayOff				:= C_5640_501_06_RTC01_SP_Tid_Stdb_R0422,
  AV_SetpointAirQuality			:= C_5640_501_06_RYA601_SP_R0422,
  AI_CurrentCo2					:= C_5640_501_06_RYA601_MV_R0422,
  AO_ControlledVariableHeating	:= C_5640_501_06_SBB01_C_R0422,
  modbusHoldingRegisters		:= ADR(GVL_Modbus.awHoldingRegisters[i * 40]), 
  modbusCoilRegisters			:= ADR(GVL_Modbus.axCoils[i]), 
  typClimateControllerInterface	:= GVL_ClimateControl.typClimateControllerInterfaceRoom422, 
  typClimateControllerSettings  := PersistentVars.typClimateControllerSettingsRoom422
);
i := i +1;
                
// Mappinger for rom 426_1

bacnetModbusClimateInterop[i](
  BO_PresenceDetection			:= C_5640_501_06_RBA01_D_R0426_1,
  AI_CurrentTemperature			:= C_5640_501_06_RTC01_MV_R0426_1,
  AV_CurrentHeatingSetpoint		:= C_5640_501_06_RTC01_SPV_R0426_1,
  AV_ComfortHeatingSetpoint		:= C_5640_501_06_RTC01_SPV_Komf_R0426_1,
  AV_StandbyHeatingSetpoint		:= C_5640_501_06_RTC01_SPV_Stdb_R0426_1,
  AV_EconomyHeatingSetpoint		:= C_5640_501_06_RTC01_SPV_Natt_R0426_1,
  MSV_CurrentWorkingMode			:= C_5640_501_06_RTC01_MOD_FB_R0426_1,
  MSV_Calendar					:= C_5640_501_06_RTC01_KMD_MSV_R0426_1,
  AV_PresenceDelayOff				:= C_5640_501_06_RTC01_SP_Tid_Stdb_R0426_1,
  AV_SetpointAirQuality			:= C_5640_501_06_RYA601_SP_R0426_1,
  AI_CurrentCo2					:= C_5640_501_06_RYA601_MV_R0426_1,
  AO_ControlledVariableHeating	:= C_5640_501_06_SBB01_C_R0426_1,
  modbusHoldingRegisters		:= ADR(GVL_Modbus.awHoldingRegisters[i * 40]), 
  modbusCoilRegisters			:= ADR(GVL_Modbus.axCoils[i]), 
  typClimateControllerInterface	:= GVL_ClimateControl.typClimateControllerInterfaceRoom426_1, 
  typClimateControllerSettings  := PersistentVars.typClimateControllerSettingsRoom426_1
);
i := i +1;
                
// Mappinger for rom 426_2

bacnetModbusClimateInterop[i](
  BO_PresenceDetection			:= C_5640_501_06_RBA01_D_R0426_2,
  AI_CurrentTemperature			:= C_5640_501_06_RTC01_MV_R0426_2,
  AV_CurrentHeatingSetpoint		:= C_5640_501_06_RTC01_SPV_R0426_2,
  AV_ComfortHeatingSetpoint		:= C_5640_501_06_RTC01_SPV_Komf_R0426_2,
  AV_StandbyHeatingSetpoint		:= C_5640_501_06_RTC01_SPV_Stdb_R0426_2,
  AV_EconomyHeatingSetpoint		:= C_5640_501_06_RTC01_SPV_Natt_R0426_2,
  MSV_CurrentWorkingMode			:= C_5640_501_06_RTC01_MOD_FB_R0426_2,
  MSV_Calendar					:= C_5640_501_06_RTC01_KMD_MSV_R0426_2,
  AV_PresenceDelayOff				:= C_5640_501_06_RTC01_SP_Tid_Stdb_R0426_2,
  AV_SetpointAirQuality			:= C_5640_501_06_RYA601_SP_R0426_2,
  AI_CurrentCo2					:= C_5640_501_06_RYA601_MV_R0426_2,
  AO_ControlledVariableHeating	:= C_5640_501_06_SBB01_C_R0426_2,
  modbusHoldingRegisters		:= ADR(GVL_Modbus.awHoldingRegisters[i * 40]), 
  modbusCoilRegisters			:= ADR(GVL_Modbus.axCoils[i]), 
  typClimateControllerInterface	:= GVL_ClimateControl.typClimateControllerInterfaceRoom426_2, 
  typClimateControllerSettings  := PersistentVars.typClimateControllerSettingsRoom426_2
);
i := i +1;
                
// Mappinger for rom 426_3

bacnetModbusClimateInterop[i](
  BO_PresenceDetection			:= C_5640_501_06_RBA01_D_R0426_3,
  AI_CurrentTemperature			:= C_5640_501_06_RTC01_MV_R0426_3,
  AV_CurrentHeatingSetpoint		:= C_5640_501_06_RTC01_SPV_R0426_3,
  AV_ComfortHeatingSetpoint		:= C_5640_501_06_RTC01_SPV_Komf_R0426_3,
  AV_StandbyHeatingSetpoint		:= C_5640_501_06_RTC01_SPV_Stdb_R0426_3,
  AV_EconomyHeatingSetpoint		:= C_5640_501_06_RTC01_SPV_Natt_R0426_3,
  MSV_CurrentWorkingMode			:= C_5640_501_06_RTC01_MOD_FB_R0426_3,
  MSV_Calendar					:= C_5640_501_06_RTC01_KMD_MSV_R0426_3,
  AV_PresenceDelayOff				:= C_5640_501_06_RTC01_SP_Tid_Stdb_R0426_3,
  AV_SetpointAirQuality			:= C_5640_501_06_RYA601_SP_R0426_3,
  AI_CurrentCo2					:= C_5640_501_06_RYA601_MV_R0426_3,
  AO_ControlledVariableHeating	:= C_5640_501_06_SBB01_C_R0426_3,
  modbusHoldingRegisters		:= ADR(GVL_Modbus.awHoldingRegisters[i * 40]), 
  modbusCoilRegisters			:= ADR(GVL_Modbus.axCoils[i]), 
  typClimateControllerInterface	:= GVL_ClimateControl.typClimateControllerInterfaceRoom426_3, 
  typClimateControllerSettings  := PersistentVars.typClimateControllerSettingsRoom426_3
);
i := i +1;
                
// Mappinger for rom 528

bacnetModbusClimateInterop[i](
  BO_PresenceDetection			:= C_5640_501_06_RBA01_D_R0528,
  AI_CurrentTemperature			:= C_5640_501_06_RTC01_MV_R0528,
  AV_CurrentHeatingSetpoint		:= C_5640_501_06_RTC01_SPV_R0528,
  AV_ComfortHeatingSetpoint		:= C_5640_501_06_RTC01_SPV_Komf_R0528,
  AV_StandbyHeatingSetpoint		:= C_5640_501_06_RTC01_SPV_Stdb_R0528,
  AV_EconomyHeatingSetpoint		:= C_5640_501_06_RTC01_SPV_Natt_R0528,
  MSV_CurrentWorkingMode			:= C_5640_501_06_RTC01_MOD_FB_R0528,
  MSV_Calendar					:= C_5640_501_06_RTC01_KMD_MSV_R0528,
  AV_PresenceDelayOff				:= C_5640_501_06_RTC01_SP_Tid_Stdb_R0528,
  AV_SetpointAirQuality			:= C_5640_501_06_RYA601_SP_R0528,
  AI_CurrentCo2					:= C_5640_501_06_RYA601_MV_R0528,
  AO_ControlledVariableHeating	:= C_5640_501_06_SBB01_C_R0528,
  modbusHoldingRegisters		:= ADR(GVL_Modbus.awHoldingRegisters[i * 40]), 
  modbusCoilRegisters			:= ADR(GVL_Modbus.axCoils[i]), 
  typClimateControllerInterface	:= GVL_ClimateControl.typClimateControllerInterfaceRoom528, 
  typClimateControllerSettings  := PersistentVars.typClimateControllerSettingsRoom528
);
i := i +1;
                
// Mappinger for rom 523

bacnetModbusClimateInterop[i](
  BO_PresenceDetection			:= C_5640_501_06_RBA01_D_R0523,
  AI_CurrentTemperature			:= C_5640_501_06_RTC01_MV_R0523,
  AV_CurrentHeatingSetpoint		:= C_5640_501_06_RTC01_SPV_R0523,
  AV_ComfortHeatingSetpoint		:= C_5640_501_06_RTC01_SPV_Komf_R0523,
  AV_StandbyHeatingSetpoint		:= C_5640_501_06_RTC01_SPV_Stdb_R0523,
  AV_EconomyHeatingSetpoint		:= C_5640_501_06_RTC01_SPV_Natt_R0523,
  MSV_CurrentWorkingMode			:= C_5640_501_06_RTC01_MOD_FB_R0523,
  MSV_Calendar					:= C_5640_501_06_RTC01_KMD_MSV_R0523,
  AV_PresenceDelayOff				:= C_5640_501_06_RTC01_SP_Tid_Stdb_R0523,
  AV_SetpointAirQuality			:= C_5640_501_06_RYA601_SP_R0523,
  AI_CurrentCo2					:= C_5640_501_06_RYA601_MV_R0523,
  AO_ControlledVariableHeating	:= C_5640_501_06_SBB01_C_R0523,
  modbusHoldingRegisters		:= ADR(GVL_Modbus.awHoldingRegisters[i * 40]), 
  modbusCoilRegisters			:= ADR(GVL_Modbus.axCoils[i]), 
  typClimateControllerInterface	:= GVL_ClimateControl.typClimateControllerInterfaceRoom523, 
  typClimateControllerSettings  := PersistentVars.typClimateControllerSettingsRoom523
);
i := i +1;
                
// Mappinger for rom 531

bacnetModbusClimateInterop[i](
  BO_PresenceDetection			:= C_5640_501_06_RBA01_D_R0531,
  AI_CurrentTemperature			:= C_5640_501_06_RTC01_MV_R0531,
  AV_CurrentHeatingSetpoint		:= C_5640_501_06_RTC01_SPV_R0531,
  AV_ComfortHeatingSetpoint		:= C_5640_501_06_RTC01_SPV_Komf_R0531,
  AV_StandbyHeatingSetpoint		:= C_5640_501_06_RTC01_SPV_Stdb_R0531,
  AV_EconomyHeatingSetpoint		:= C_5640_501_06_RTC01_SPV_Natt_R0531,
  MSV_CurrentWorkingMode			:= C_5640_501_06_RTC01_MOD_FB_R0531,
  MSV_Calendar					:= C_5640_501_06_RTC01_KMD_MSV_R0531,
  AV_PresenceDelayOff				:= C_5640_501_06_RTC01_SP_Tid_Stdb_R0531,
  AV_SetpointAirQuality			:= C_5640_501_06_RYA601_SP_R0531,
  AI_CurrentCo2					:= C_5640_501_06_RYA601_MV_R0531,
  AO_ControlledVariableHeating	:= C_5640_501_06_SBB01_C_R0531,
  modbusHoldingRegisters		:= ADR(GVL_Modbus.awHoldingRegisters[i * 40]), 
  modbusCoilRegisters			:= ADR(GVL_Modbus.axCoils[i]), 
  typClimateControllerInterface	:= GVL_ClimateControl.typClimateControllerInterfaceRoom531, 
  typClimateControllerSettings  := PersistentVars.typClimateControllerSettingsRoom531
);
i := i +1;
                
// Mappinger for rom 535_1

bacnetModbusClimateInterop[i](
  BO_PresenceDetection			:= C_5640_501_06_RBA01_D_R0535_1,
  AI_CurrentTemperature			:= C_5640_501_06_RTC01_MV_R0535_1,
  AV_CurrentHeatingSetpoint		:= C_5640_501_06_RTC01_SPV_R0535_1,
  AV_ComfortHeatingSetpoint		:= C_5640_501_06_RTC01_SPV_Komf_R0535_1,
  AV_StandbyHeatingSetpoint		:= C_5640_501_06_RTC01_SPV_Stdb_R0535_1,
  AV_EconomyHeatingSetpoint		:= C_5640_501_06_RTC01_SPV_Natt_R0535_1,
  MSV_CurrentWorkingMode			:= C_5640_501_06_RTC01_MOD_FB_R0535_1,
  MSV_Calendar					:= C_5640_501_06_RTC01_KMD_MSV_R0535_1,
  AV_PresenceDelayOff				:= C_5640_501_06_RTC01_SP_Tid_Stdb_R0535_1,
  AV_SetpointAirQuality			:= C_5640_501_06_RYA601_SP_R0535_1,
  AI_CurrentCo2					:= C_5640_501_06_RYA601_MV_R0535_1,
  AO_ControlledVariableHeating	:= C_5640_501_06_SBB01_C_R0535_1,
  modbusHoldingRegisters		:= ADR(GVL_Modbus.awHoldingRegisters[i * 40]), 
  modbusCoilRegisters			:= ADR(GVL_Modbus.axCoils[i]), 
  typClimateControllerInterface	:= GVL_ClimateControl.typClimateControllerInterfaceRoom535_1, 
  typClimateControllerSettings  := PersistentVars.typClimateControllerSettingsRoom535_1
);
i := i +1;
                
// Mappinger for rom 535_2

bacnetModbusClimateInterop[i](
  BO_PresenceDetection			:= C_5640_501_06_RBA01_D_R0535_2,
  AI_CurrentTemperature			:= C_5640_501_06_RTC01_MV_R0535_2,
  AV_CurrentHeatingSetpoint		:= C_5640_501_06_RTC01_SPV_R0535_2,
  AV_ComfortHeatingSetpoint		:= C_5640_501_06_RTC01_SPV_Komf_R0535_2,
  AV_StandbyHeatingSetpoint		:= C_5640_501_06_RTC01_SPV_Stdb_R0535_2,
  AV_EconomyHeatingSetpoint		:= C_5640_501_06_RTC01_SPV_Natt_R0535_2,
  MSV_CurrentWorkingMode			:= C_5640_501_06_RTC01_MOD_FB_R0535_2,
  MSV_Calendar					:= C_5640_501_06_RTC01_KMD_MSV_R0535_2,
  AV_PresenceDelayOff				:= C_5640_501_06_RTC01_SP_Tid_Stdb_R0535_2,
  AV_SetpointAirQuality			:= C_5640_501_06_RYA601_SP_R0535_2,
  AI_CurrentCo2					:= C_5640_501_06_RYA601_MV_R0535_2,
  AO_ControlledVariableHeating	:= C_5640_501_06_SBB01_C_R0535_2,
  modbusHoldingRegisters		:= ADR(GVL_Modbus.awHoldingRegisters[i * 40]), 
  modbusCoilRegisters			:= ADR(GVL_Modbus.axCoils[i]), 
  typClimateControllerInterface	:= GVL_ClimateControl.typClimateControllerInterfaceRoom535_2, 
  typClimateControllerSettings  := PersistentVars.typClimateControllerSettingsRoom535_2
);
i := i +1;
                
// Mappinger for rom 535_3

bacnetModbusClimateInterop[i](
  BO_PresenceDetection			:= C_5640_501_06_RBA01_D_R0535_3,
  AI_CurrentTemperature			:= C_5640_501_06_RTC01_MV_R0535_3,
  AV_CurrentHeatingSetpoint		:= C_5640_501_06_RTC01_SPV_R0535_3,
  AV_ComfortHeatingSetpoint		:= C_5640_501_06_RTC01_SPV_Komf_R0535_3,
  AV_StandbyHeatingSetpoint		:= C_5640_501_06_RTC01_SPV_Stdb_R0535_3,
  AV_EconomyHeatingSetpoint		:= C_5640_501_06_RTC01_SPV_Natt_R0535_3,
  MSV_CurrentWorkingMode			:= C_5640_501_06_RTC01_MOD_FB_R0535_3,
  MSV_Calendar					:= C_5640_501_06_RTC01_KMD_MSV_R0535_3,
  AV_PresenceDelayOff				:= C_5640_501_06_RTC01_SP_Tid_Stdb_R0535_3,
  AV_SetpointAirQuality			:= C_5640_501_06_RYA601_SP_R0535_3,
  AI_CurrentCo2					:= C_5640_501_06_RYA601_MV_R0535_3,
  AO_ControlledVariableHeating	:= C_5640_501_06_SBB01_C_R0535_3,
  modbusHoldingRegisters		:= ADR(GVL_Modbus.awHoldingRegisters[i * 40]), 
  modbusCoilRegisters			:= ADR(GVL_Modbus.axCoils[i]), 
  typClimateControllerInterface	:= GVL_ClimateControl.typClimateControllerInterfaceRoom535_3, 
  typClimateControllerSettings  := PersistentVars.typClimateControllerSettingsRoom535_3
);
i := i +1;
                
// Mappinger for rom 536

bacnetModbusClimateInterop[i](
  BO_PresenceDetection			:= C_5640_501_06_RBA01_D_R0536,
  AI_CurrentTemperature			:= C_5640_501_06_RTC01_MV_R0536,
  AV_CurrentHeatingSetpoint		:= C_5640_501_06_RTC01_SPV_R0536,
  AV_ComfortHeatingSetpoint		:= C_5640_501_06_RTC01_SPV_Komf_R0536,
  AV_StandbyHeatingSetpoint		:= C_5640_501_06_RTC01_SPV_Stdb_R0536,
  AV_EconomyHeatingSetpoint		:= C_5640_501_06_RTC01_SPV_Natt_R0536,
  MSV_CurrentWorkingMode			:= C_5640_501_06_RTC01_MOD_FB_R0536,
  MSV_Calendar					:= C_5640_501_06_RTC01_KMD_MSV_R0536,
  AV_PresenceDelayOff				:= C_5640_501_06_RTC01_SP_Tid_Stdb_R0536,
  AV_SetpointAirQuality			:= C_5640_501_06_RYA601_SP_R0536,
  AI_CurrentCo2					:= C_5640_501_06_RYA601_MV_R0536,
  AO_ControlledVariableHeating	:= C_5640_501_06_SBB01_C_R0536,
  modbusHoldingRegisters		:= ADR(GVL_Modbus.awHoldingRegisters[i * 40]), 
  modbusCoilRegisters			:= ADR(GVL_Modbus.axCoils[i]), 
  typClimateControllerInterface	:= GVL_ClimateControl.typClimateControllerInterfaceRoom536, 
  typClimateControllerSettings  := PersistentVars.typClimateControllerSettingsRoom536
);
i := i +1;
                
// Mappinger for rom 543

bacnetModbusClimateInterop[i](
  BO_PresenceDetection			:= C_5640_501_06_RBA01_D_R0543,
  AI_CurrentTemperature			:= C_5640_501_06_RTC01_MV_R0543,
  AV_CurrentHeatingSetpoint		:= C_5640_501_06_RTC01_SPV_R0543,
  AV_ComfortHeatingSetpoint		:= C_5640_501_06_RTC01_SPV_Komf_R0543,
  AV_StandbyHeatingSetpoint		:= C_5640_501_06_RTC01_SPV_Stdb_R0543,
  AV_EconomyHeatingSetpoint		:= C_5640_501_06_RTC01_SPV_Natt_R0543,
  MSV_CurrentWorkingMode			:= C_5640_501_06_RTC01_MOD_FB_R0543,
  MSV_Calendar					:= C_5640_501_06_RTC01_KMD_MSV_R0543,
  AV_PresenceDelayOff				:= C_5640_501_06_RTC01_SP_Tid_Stdb_R0543,
  AV_SetpointAirQuality			:= C_5640_501_06_RYA601_SP_R0543,
  AI_CurrentCo2					:= C_5640_501_06_RYA601_MV_R0543,
  AO_ControlledVariableHeating	:= C_5640_501_06_SBB01_C_R0543,
  modbusHoldingRegisters		:= ADR(GVL_Modbus.awHoldingRegisters[i * 40]), 
  modbusCoilRegisters			:= ADR(GVL_Modbus.axCoils[i]), 
  typClimateControllerInterface	:= GVL_ClimateControl.typClimateControllerInterfaceRoom543, 
  typClimateControllerSettings  := PersistentVars.typClimateControllerSettingsRoom543
);
i := i +1;
                
// Mappinger for rom 547_1

bacnetModbusClimateInterop[i](
  BO_PresenceDetection			:= C_5640_501_06_RBA01_D_R0547_1,
  AI_CurrentTemperature			:= C_5640_501_06_RTC01_MV_R0547_1,
  AV_CurrentHeatingSetpoint		:= C_5640_501_06_RTC01_SPV_R0547_1,
  AV_ComfortHeatingSetpoint		:= C_5640_501_06_RTC01_SPV_Komf_R0547_1,
  AV_StandbyHeatingSetpoint		:= C_5640_501_06_RTC01_SPV_Stdb_R0547_1,
  AV_EconomyHeatingSetpoint		:= C_5640_501_06_RTC01_SPV_Natt_R0547_1,
  MSV_CurrentWorkingMode			:= C_5640_501_06_RTC01_MOD_FB_R0547_1,
  MSV_Calendar					:= C_5640_501_06_RTC01_KMD_MSV_R0547_1,
  AV_PresenceDelayOff				:= C_5640_501_06_RTC01_SP_Tid_Stdb_R0547_1,
  AV_SetpointAirQuality			:= C_5640_501_06_RYA601_SP_R0547_1,
  AI_CurrentCo2					:= C_5640_501_06_RYA601_MV_R0547_1,
  AO_ControlledVariableHeating	:= C_5640_501_06_SBB01_C_R0547_1,
  modbusHoldingRegisters		:= ADR(GVL_Modbus.awHoldingRegisters[i * 40]), 
  modbusCoilRegisters			:= ADR(GVL_Modbus.axCoils[i]), 
  typClimateControllerInterface	:= GVL_ClimateControl.typClimateControllerInterfaceRoom547_1, 
  typClimateControllerSettings  := PersistentVars.typClimateControllerSettingsRoom547_1
);
i := i +1;
                
// Mappinger for rom 547_2

bacnetModbusClimateInterop[i](
  BO_PresenceDetection			:= C_5640_501_06_RBA01_D_R0547_2,
  AI_CurrentTemperature			:= C_5640_501_06_RTC01_MV_R0547_2,
  AV_CurrentHeatingSetpoint		:= C_5640_501_06_RTC01_SPV_R0547_2,
  AV_ComfortHeatingSetpoint		:= C_5640_501_06_RTC01_SPV_Komf_R0547_2,
  AV_StandbyHeatingSetpoint		:= C_5640_501_06_RTC01_SPV_Stdb_R0547_2,
  AV_EconomyHeatingSetpoint		:= C_5640_501_06_RTC01_SPV_Natt_R0547_2,
  MSV_CurrentWorkingMode			:= C_5640_501_06_RTC01_MOD_FB_R0547_2,
  MSV_Calendar					:= C_5640_501_06_RTC01_KMD_MSV_R0547_2,
  AV_PresenceDelayOff				:= C_5640_501_06_RTC01_SP_Tid_Stdb_R0547_2,
  AV_SetpointAirQuality			:= C_5640_501_06_RYA601_SP_R0547_2,
  AI_CurrentCo2					:= C_5640_501_06_RYA601_MV_R0547_2,
  AO_ControlledVariableHeating	:= C_5640_501_06_SBB01_C_R0547_2,
  modbusHoldingRegisters		:= ADR(GVL_Modbus.awHoldingRegisters[i * 40]), 
  modbusCoilRegisters			:= ADR(GVL_Modbus.axCoils[i]), 
  typClimateControllerInterface	:= GVL_ClimateControl.typClimateControllerInterfaceRoom547_2, 
  typClimateControllerSettings  := PersistentVars.typClimateControllerSettingsRoom547_2
);
i := i +1;
                
// Mappinger for rom 544

bacnetModbusClimateInterop[i](
  BO_PresenceDetection			:= C_5640_501_06_RBA01_D_R0544,
  AI_CurrentTemperature			:= C_5640_501_06_RTC01_MV_R0544,
  AV_CurrentHeatingSetpoint		:= C_5640_501_06_RTC01_SPV_R0544,
  AV_ComfortHeatingSetpoint		:= C_5640_501_06_RTC01_SPV_Komf_R0544,
  AV_StandbyHeatingSetpoint		:= C_5640_501_06_RTC01_SPV_Stdb_R0544,
  AV_EconomyHeatingSetpoint		:= C_5640_501_06_RTC01_SPV_Natt_R0544,
  MSV_CurrentWorkingMode			:= C_5640_501_06_RTC01_MOD_FB_R0544,
  MSV_Calendar					:= C_5640_501_06_RTC01_KMD_MSV_R0544,
  AV_PresenceDelayOff				:= C_5640_501_06_RTC01_SP_Tid_Stdb_R0544,
  AV_SetpointAirQuality			:= C_5640_501_06_RYA601_SP_R0544,
  AI_CurrentCo2					:= C_5640_501_06_RYA601_MV_R0544,
  AO_ControlledVariableHeating	:= C_5640_501_06_SBB01_C_R0544,
  modbusHoldingRegisters		:= ADR(GVL_Modbus.awHoldingRegisters[i * 40]), 
  modbusCoilRegisters			:= ADR(GVL_Modbus.axCoils[i]), 
  typClimateControllerInterface	:= GVL_ClimateControl.typClimateControllerInterfaceRoom544, 
  typClimateControllerSettings  := PersistentVars.typClimateControllerSettingsRoom544
);
i := i +1;
i := 50;

                
// Mappinger for spjeld +A=360.01-SQ4A407

bacnetModbusDamperInterop[1][1](
  AI_Volume					:= A_360_01_SQ4_A407_VOL,
  AV_CurrentSetpoint			:= A_360_01_SQ4_A407_SP,
  AV_vMin					:= A_360_01_SQ4_A407_VMIN,
  AV_vMax					:= A_360_01_SQ4_A407_VMAX,
  AI_Position				:= A_360_01_SQ4_A407_FB,
  AV_ControlledVariable		:= A_360_01_SQ4_A407_C,
  AV_ManualOverride			:= A_360_01_SQ4_A407_KMD,
  BV_ExcludeFromOptimizer	:= A_360_01_SQ4_A407_OPT_EKSKL,
  BV_DamperError				:= A_360_01_SQ4_A407_A1,
  BV_CommunicationError		:= A_360_01_SQ4_A407_A2,
  modbusHoldingRegisters		:= ADR(GVL_Modbus.awHoldingRegisters[i * 30]), 
  modbusCoilRegisters			:= ADR(GVL_Modbus.axCoils[i]), 
  typDamperInterface	    :=  GVL_Modbus.ModbusDamperInterface[1][1], 
  typDamperSettings       := PersistentVars.ModbusDamperSetpoints[1][1]
);
i := i +1;
// Kommunikasjonsalarmer

                
// Mappinger for spjeld +A=360.01-SQ44AH2

bacnetModbusDamperInterop[1][2](
  AI_Volume					:= A_360_01_SQ4_4AH2_VOL,
  AV_CurrentSetpoint			:= A_360_01_SQ4_4AH2_SP,
  AV_vMin					:= A_360_01_SQ4_4AH2_VMIN,
  AV_vMax					:= A_360_01_SQ4_4AH2_VMAX,
  AI_Position				:= A_360_01_SQ4_4AH2_FB,
  AV_ControlledVariable		:= A_360_01_SQ4_4AH2_C,
  AV_ManualOverride			:= A_360_01_SQ4_4AH2_KMD,
  BV_ExcludeFromOptimizer	:= A_360_01_SQ4_4AH2_OPT_EKSKL,
  BV_DamperError				:= A_360_01_SQ4_4AH2_A1,
  BV_CommunicationError		:= A_360_01_SQ4_4AH2_A2,
  modbusHoldingRegisters		:= ADR(GVL_Modbus.awHoldingRegisters[i * 30]), 
  modbusCoilRegisters			:= ADR(GVL_Modbus.axCoils[i]), 
  typDamperInterface	    :=  GVL_Modbus.ModbusDamperInterface[1][2], 
  typDamperSettings       := PersistentVars.ModbusDamperSetpoints[1][2]
);
i := i +1;
// Kommunikasjonsalarmer

                
// Mappinger for spjeld +A=360.01-SQ44AH1

bacnetModbusDamperInterop[1][3](
  AI_Volume					:= A_360_01_SQ4_4AH1_VOL,
  AV_CurrentSetpoint			:= A_360_01_SQ4_4AH1_SP,
  AV_vMin					:= A_360_01_SQ4_4AH1_VMIN,
  AV_vMax					:= A_360_01_SQ4_4AH1_VMAX,
  AI_Position				:= A_360_01_SQ4_4AH1_FB,
  AV_ControlledVariable		:= A_360_01_SQ4_4AH1_C,
  AV_ManualOverride			:= A_360_01_SQ4_4AH1_KMD,
  BV_ExcludeFromOptimizer	:= A_360_01_SQ4_4AH1_OPT_EKSKL,
  BV_DamperError				:= A_360_01_SQ4_4AH1_A1,
  BV_CommunicationError		:= A_360_01_SQ4_4AH1_A2,
  modbusHoldingRegisters		:= ADR(GVL_Modbus.awHoldingRegisters[i * 30]), 
  modbusCoilRegisters			:= ADR(GVL_Modbus.axCoils[i]), 
  typDamperInterface	    :=  GVL_Modbus.ModbusDamperInterface[1][3], 
  typDamperSettings       := PersistentVars.ModbusDamperSetpoints[1][3]
);
i := i +1;
// Kommunikasjonsalarmer

                
// Mappinger for spjeld +A=360.01-SQ54AH1

bacnetModbusDamperInterop[1][4](
  AI_Volume					:= A_360_01_SQ5_4AH1_VOL,
  AV_CurrentSetpoint			:= A_360_01_SQ5_4AH1_SP,
  AV_vMin					:= A_360_01_SQ5_4AH1_VMIN,
  AV_vMax					:= A_360_01_SQ5_4AH1_VMAX,
  AI_Position				:= A_360_01_SQ5_4AH1_FB,
  AV_ControlledVariable		:= A_360_01_SQ5_4AH1_C,
  AV_ManualOverride			:= A_360_01_SQ5_4AH1_KMD,
  BV_ExcludeFromOptimizer	:= A_360_01_SQ5_4AH1_OPT_EKSKL,
  BV_DamperError				:= A_360_01_SQ5_4AH1_A1,
  BV_CommunicationError		:= A_360_01_SQ5_4AH1_A2,
  modbusHoldingRegisters		:= ADR(GVL_Modbus.awHoldingRegisters[i * 30]), 
  modbusCoilRegisters			:= ADR(GVL_Modbus.axCoils[i]), 
  typDamperInterface	    :=  GVL_Modbus.ModbusDamperInterface[1][4], 
  typDamperSettings       := PersistentVars.ModbusDamperSetpoints[1][4]
);
i := i +1;
// Kommunikasjonsalarmer

                
// Mappinger for spjeld +A=360.01-SQ5A405

bacnetModbusDamperInterop[1][5](
  AI_Volume					:= A_360_01_SQ5_A405_VOL,
  AV_CurrentSetpoint			:= A_360_01_SQ5_A405_SP,
  AV_vMin					:= A_360_01_SQ5_A405_VMIN,
  AV_vMax					:= A_360_01_SQ5_A405_VMAX,
  AI_Position				:= A_360_01_SQ5_A405_FB,
  AV_ControlledVariable		:= A_360_01_SQ5_A405_C,
  AV_ManualOverride			:= A_360_01_SQ5_A405_KMD,
  BV_ExcludeFromOptimizer	:= A_360_01_SQ5_A405_OPT_EKSKL,
  BV_DamperError				:= A_360_01_SQ5_A405_A1,
  BV_CommunicationError		:= A_360_01_SQ5_A405_A2,
  modbusHoldingRegisters		:= ADR(GVL_Modbus.awHoldingRegisters[i * 30]), 
  modbusCoilRegisters			:= ADR(GVL_Modbus.axCoils[i]), 
  typDamperInterface	    :=  GVL_Modbus.ModbusDamperInterface[1][5], 
  typDamperSettings       := PersistentVars.ModbusDamperSetpoints[1][5]
);
i := i +1;
// Kommunikasjonsalarmer

                
// Mappinger for spjeld +A=360.01-SQ4A401_2

bacnetModbusDamperInterop[1][6](
  AI_Volume					:= A_360_01_SQ4_A401_2_VOL,
  AV_CurrentSetpoint			:= A_360_01_SQ4_A401_2_SP,
  AV_vMin					:= A_360_01_SQ4_A401_2_VMIN,
  AV_vMax					:= A_360_01_SQ4_A401_2_VMAX,
  AI_Position				:= A_360_01_SQ4_A401_2_FB,
  AV_ControlledVariable		:= A_360_01_SQ4_A401_2_C,
  AV_ManualOverride			:= A_360_01_SQ4_A401_2_KMD,
  BV_ExcludeFromOptimizer	:= A_360_01_SQ4_A401_2_OPT_EKSKL,
  BV_DamperError				:= A_360_01_SQ4_A401_2_A1,
  BV_CommunicationError		:= A_360_01_SQ4_A401_2_A2,
  modbusHoldingRegisters		:= ADR(GVL_Modbus.awHoldingRegisters[i * 30]), 
  modbusCoilRegisters			:= ADR(GVL_Modbus.axCoils[i]), 
  typDamperInterface	    :=  GVL_Modbus.ModbusDamperInterface[1][6], 
  typDamperSettings       := PersistentVars.ModbusDamperSetpoints[1][6]
);
i := i +1;
// Kommunikasjonsalarmer

                
// Mappinger for spjeld +A=360.01-SQ4A401_1

bacnetModbusDamperInterop[1][7](
  AI_Volume					:= A_360_01_SQ4_A401_1_VOL,
  AV_CurrentSetpoint			:= A_360_01_SQ4_A401_1_SP,
  AV_vMin					:= A_360_01_SQ4_A401_1_VMIN,
  AV_vMax					:= A_360_01_SQ4_A401_1_VMAX,
  AI_Position				:= A_360_01_SQ4_A401_1_FB,
  AV_ControlledVariable		:= A_360_01_SQ4_A401_1_C,
  AV_ManualOverride			:= A_360_01_SQ4_A401_1_KMD,
  BV_ExcludeFromOptimizer	:= A_360_01_SQ4_A401_1_OPT_EKSKL,
  BV_DamperError				:= A_360_01_SQ4_A401_1_A1,
  BV_CommunicationError		:= A_360_01_SQ4_A401_1_A2,
  modbusHoldingRegisters		:= ADR(GVL_Modbus.awHoldingRegisters[i * 30]), 
  modbusCoilRegisters			:= ADR(GVL_Modbus.axCoils[i]), 
  typDamperInterface	    :=  GVL_Modbus.ModbusDamperInterface[1][7], 
  typDamperSettings       := PersistentVars.ModbusDamperSetpoints[1][7]
);
i := i +1;
// Kommunikasjonsalarmer

                
// Mappinger for spjeld +A=360.01-SQ4A401

bacnetModbusDamperInterop[1][8](
  AI_Volume					:= A_360_01_SQ4_A401_VOL,
  AV_CurrentSetpoint			:= A_360_01_SQ4_A401_SP,
  AV_vMin					:= A_360_01_SQ4_A401_VMIN,
  AV_vMax					:= A_360_01_SQ4_A401_VMAX,
  AI_Position				:= A_360_01_SQ4_A401_FB,
  AV_ControlledVariable		:= A_360_01_SQ4_A401_C,
  AV_ManualOverride			:= A_360_01_SQ4_A401_KMD,
  BV_ExcludeFromOptimizer	:= A_360_01_SQ4_A401_OPT_EKSKL,
  BV_DamperError				:= A_360_01_SQ4_A401_A1,
  BV_CommunicationError		:= A_360_01_SQ4_A401_A2,
  modbusHoldingRegisters		:= ADR(GVL_Modbus.awHoldingRegisters[i * 30]), 
  modbusCoilRegisters			:= ADR(GVL_Modbus.axCoils[i]), 
  typDamperInterface	    :=  GVL_Modbus.ModbusDamperInterface[1][8], 
  typDamperSettings       := PersistentVars.ModbusDamperSetpoints[1][8]
);
i := i +1;
// Kommunikasjonsalarmer

                
// Mappinger for spjeld +A=360.01-SQ4A406

bacnetModbusDamperInterop[1][9](
  AI_Volume					:= A_360_01_SQ4_A406_VOL,
  AV_CurrentSetpoint			:= A_360_01_SQ4_A406_SP,
  AV_vMin					:= A_360_01_SQ4_A406_VMIN,
  AV_vMax					:= A_360_01_SQ4_A406_VMAX,
  AI_Position				:= A_360_01_SQ4_A406_FB,
  AV_ControlledVariable		:= A_360_01_SQ4_A406_C,
  AV_ManualOverride			:= A_360_01_SQ4_A406_KMD,
  BV_ExcludeFromOptimizer	:= A_360_01_SQ4_A406_OPT_EKSKL,
  BV_DamperError				:= A_360_01_SQ4_A406_A1,
  BV_CommunicationError		:= A_360_01_SQ4_A406_A2,
  modbusHoldingRegisters		:= ADR(GVL_Modbus.awHoldingRegisters[i * 30]), 
  modbusCoilRegisters			:= ADR(GVL_Modbus.axCoils[i]), 
  typDamperInterface	    :=  GVL_Modbus.ModbusDamperInterface[1][9], 
  typDamperSettings       := PersistentVars.ModbusDamperSetpoints[1][9]
);
i := i +1;
// Kommunikasjonsalarmer

                
// Mappinger for spjeld +A=360.01-SQ4A408

bacnetModbusDamperInterop[1][10](
  AI_Volume					:= A_360_01_SQ4_A408_VOL,
  AV_CurrentSetpoint			:= A_360_01_SQ4_A408_SP,
  AV_vMin					:= A_360_01_SQ4_A408_VMIN,
  AV_vMax					:= A_360_01_SQ4_A408_VMAX,
  AI_Position				:= A_360_01_SQ4_A408_FB,
  AV_ControlledVariable		:= A_360_01_SQ4_A408_C,
  AV_ManualOverride			:= A_360_01_SQ4_A408_KMD,
  BV_ExcludeFromOptimizer	:= A_360_01_SQ4_A408_OPT_EKSKL,
  BV_DamperError				:= A_360_01_SQ4_A408_A1,
  BV_CommunicationError		:= A_360_01_SQ4_A408_A2,
  modbusHoldingRegisters		:= ADR(GVL_Modbus.awHoldingRegisters[i * 30]), 
  modbusCoilRegisters			:= ADR(GVL_Modbus.axCoils[i]), 
  typDamperInterface	    :=  GVL_Modbus.ModbusDamperInterface[1][10], 
  typDamperSettings       := PersistentVars.ModbusDamperSetpoints[1][10]
);
i := i +1;
// Kommunikasjonsalarmer

                
// Mappinger for spjeld +A=360.01-SQ4A410_1

bacnetModbusDamperInterop[1][11](
  AI_Volume					:= A_360_01_SQ4_A410_1_VOL,
  AV_CurrentSetpoint			:= A_360_01_SQ4_A410_1_SP,
  AV_vMin					:= A_360_01_SQ4_A410_1_VMIN,
  AV_vMax					:= A_360_01_SQ4_A410_1_VMAX,
  AI_Position				:= A_360_01_SQ4_A410_1_FB,
  AV_ControlledVariable		:= A_360_01_SQ4_A410_1_C,
  AV_ManualOverride			:= A_360_01_SQ4_A410_1_KMD,
  BV_ExcludeFromOptimizer	:= A_360_01_SQ4_A410_1_OPT_EKSKL,
  BV_DamperError				:= A_360_01_SQ4_A410_1_A1,
  BV_CommunicationError		:= A_360_01_SQ4_A410_1_A2,
  modbusHoldingRegisters		:= ADR(GVL_Modbus.awHoldingRegisters[i * 30]), 
  modbusCoilRegisters			:= ADR(GVL_Modbus.axCoils[i]), 
  typDamperInterface	    :=  GVL_Modbus.ModbusDamperInterface[1][11], 
  typDamperSettings       := PersistentVars.ModbusDamperSetpoints[1][11]
);
i := i +1;
// Kommunikasjonsalarmer

                
// Mappinger for spjeld +A=360.01-SQ4A410_2

bacnetModbusDamperInterop[1][12](
  AI_Volume					:= A_360_01_SQ4_A410_2_VOL,
  AV_CurrentSetpoint			:= A_360_01_SQ4_A410_2_SP,
  AV_vMin					:= A_360_01_SQ4_A410_2_VMIN,
  AV_vMax					:= A_360_01_SQ4_A410_2_VMAX,
  AI_Position				:= A_360_01_SQ4_A410_2_FB,
  AV_ControlledVariable		:= A_360_01_SQ4_A410_2_C,
  AV_ManualOverride			:= A_360_01_SQ4_A410_2_KMD,
  BV_ExcludeFromOptimizer	:= A_360_01_SQ4_A410_2_OPT_EKSKL,
  BV_DamperError				:= A_360_01_SQ4_A410_2_A1,
  BV_CommunicationError		:= A_360_01_SQ4_A410_2_A2,
  modbusHoldingRegisters		:= ADR(GVL_Modbus.awHoldingRegisters[i * 30]), 
  modbusCoilRegisters			:= ADR(GVL_Modbus.axCoils[i]), 
  typDamperInterface	    :=  GVL_Modbus.ModbusDamperInterface[1][12], 
  typDamperSettings       := PersistentVars.ModbusDamperSetpoints[1][12]
);
i := i +1;
// Kommunikasjonsalarmer

                
// Mappinger for spjeld +A=360.01-SQ4A410_3

bacnetModbusDamperInterop[1][13](
  AI_Volume					:= A_360_01_SQ4_A410_3_VOL,
  AV_CurrentSetpoint			:= A_360_01_SQ4_A410_3_SP,
  AV_vMin					:= A_360_01_SQ4_A410_3_VMIN,
  AV_vMax					:= A_360_01_SQ4_A410_3_VMAX,
  AI_Position				:= A_360_01_SQ4_A410_3_FB,
  AV_ControlledVariable		:= A_360_01_SQ4_A410_3_C,
  AV_ManualOverride			:= A_360_01_SQ4_A410_3_KMD,
  BV_ExcludeFromOptimizer	:= A_360_01_SQ4_A410_3_OPT_EKSKL,
  BV_DamperError				:= A_360_01_SQ4_A410_3_A1,
  BV_CommunicationError		:= A_360_01_SQ4_A410_3_A2,
  modbusHoldingRegisters		:= ADR(GVL_Modbus.awHoldingRegisters[i * 30]), 
  modbusCoilRegisters			:= ADR(GVL_Modbus.axCoils[i]), 
  typDamperInterface	    :=  GVL_Modbus.ModbusDamperInterface[1][13], 
  typDamperSettings       := PersistentVars.ModbusDamperSetpoints[1][13]
);
i := i +1;
// Kommunikasjonsalarmer

                
// Mappinger for spjeld +A=360.01-SQ4A410_4

bacnetModbusDamperInterop[1][14](
  AI_Volume					:= A_360_01_SQ4_A410_4_VOL,
  AV_CurrentSetpoint			:= A_360_01_SQ4_A410_4_SP,
  AV_vMin					:= A_360_01_SQ4_A410_4_VMIN,
  AV_vMax					:= A_360_01_SQ4_A410_4_VMAX,
  AI_Position				:= A_360_01_SQ4_A410_4_FB,
  AV_ControlledVariable		:= A_360_01_SQ4_A410_4_C,
  AV_ManualOverride			:= A_360_01_SQ4_A410_4_KMD,
  BV_ExcludeFromOptimizer	:= A_360_01_SQ4_A410_4_OPT_EKSKL,
  BV_DamperError				:= A_360_01_SQ4_A410_4_A1,
  BV_CommunicationError		:= A_360_01_SQ4_A410_4_A2,
  modbusHoldingRegisters		:= ADR(GVL_Modbus.awHoldingRegisters[i * 30]), 
  modbusCoilRegisters			:= ADR(GVL_Modbus.axCoils[i]), 
  typDamperInterface	    :=  GVL_Modbus.ModbusDamperInterface[1][14], 
  typDamperSettings       := PersistentVars.ModbusDamperSetpoints[1][14]
);
i := i +1;
// Kommunikasjonsalarmer

                
// Mappinger for spjeld +A=360.01-SQ4A410_5

bacnetModbusDamperInterop[1][15](
  AI_Volume					:= A_360_01_SQ4_A410_5_VOL,
  AV_CurrentSetpoint			:= A_360_01_SQ4_A410_5_SP,
  AV_vMin					:= A_360_01_SQ4_A410_5_VMIN,
  AV_vMax					:= A_360_01_SQ4_A410_5_VMAX,
  AI_Position				:= A_360_01_SQ4_A410_5_FB,
  AV_ControlledVariable		:= A_360_01_SQ4_A410_5_C,
  AV_ManualOverride			:= A_360_01_SQ4_A410_5_KMD,
  BV_ExcludeFromOptimizer	:= A_360_01_SQ4_A410_5_OPT_EKSKL,
  BV_DamperError				:= A_360_01_SQ4_A410_5_A1,
  BV_CommunicationError		:= A_360_01_SQ4_A410_5_A2,
  modbusHoldingRegisters		:= ADR(GVL_Modbus.awHoldingRegisters[i * 30]), 
  modbusCoilRegisters			:= ADR(GVL_Modbus.axCoils[i]), 
  typDamperInterface	    :=  GVL_Modbus.ModbusDamperInterface[1][15], 
  typDamperSettings       := PersistentVars.ModbusDamperSetpoints[1][15]
);
i := i +1;
// Kommunikasjonsalarmer

                
// Mappinger for spjeld +A=360.01-SQ4A412

bacnetModbusDamperInterop[1][16](
  AI_Volume					:= A_360_01_SQ4_A412_VOL,
  AV_CurrentSetpoint			:= A_360_01_SQ4_A412_SP,
  AV_vMin					:= A_360_01_SQ4_A412_VMIN,
  AV_vMax					:= A_360_01_SQ4_A412_VMAX,
  AI_Position				:= A_360_01_SQ4_A412_FB,
  AV_ControlledVariable		:= A_360_01_SQ4_A412_C,
  AV_ManualOverride			:= A_360_01_SQ4_A412_KMD,
  BV_ExcludeFromOptimizer	:= A_360_01_SQ4_A412_OPT_EKSKL,
  BV_DamperError				:= A_360_01_SQ4_A412_A1,
  BV_CommunicationError		:= A_360_01_SQ4_A412_A2,
  modbusHoldingRegisters		:= ADR(GVL_Modbus.awHoldingRegisters[i * 30]), 
  modbusCoilRegisters			:= ADR(GVL_Modbus.axCoils[i]), 
  typDamperInterface	    :=  GVL_Modbus.ModbusDamperInterface[1][16], 
  typDamperSettings       := PersistentVars.ModbusDamperSetpoints[1][16]
);
i := i +1;
// Kommunikasjonsalarmer

                
// Mappinger for spjeld +A=360.01-SQ4A413

bacnetModbusDamperInterop[1][17](
  AI_Volume					:= A_360_01_SQ4_A413_VOL,
  AV_CurrentSetpoint			:= A_360_01_SQ4_A413_SP,
  AV_vMin					:= A_360_01_SQ4_A413_VMIN,
  AV_vMax					:= A_360_01_SQ4_A413_VMAX,
  AI_Position				:= A_360_01_SQ4_A413_FB,
  AV_ControlledVariable		:= A_360_01_SQ4_A413_C,
  AV_ManualOverride			:= A_360_01_SQ4_A413_KMD,
  BV_ExcludeFromOptimizer	:= A_360_01_SQ4_A413_OPT_EKSKL,
  BV_DamperError				:= A_360_01_SQ4_A413_A1,
  BV_CommunicationError		:= A_360_01_SQ4_A413_A2,
  modbusHoldingRegisters		:= ADR(GVL_Modbus.awHoldingRegisters[i * 30]), 
  modbusCoilRegisters			:= ADR(GVL_Modbus.axCoils[i]), 
  typDamperInterface	    :=  GVL_Modbus.ModbusDamperInterface[1][17], 
  typDamperSettings       := PersistentVars.ModbusDamperSetpoints[1][17]
);
i := i +1;
// Kommunikasjonsalarmer

                
// Mappinger for spjeld +A=360.01-SK4A415

bacnetModbusDamperInterop[1][18](
  AI_Volume					:= A_360_01_SK4_A415_VOL,
  AV_CurrentSetpoint			:= A_360_01_SK4_A415_SP,
  AV_vMin					:= A_360_01_SK4_A415_VMIN,
  AV_vMax					:= A_360_01_SK4_A415_VMAX,
  AI_Position				:= A_360_01_SK4_A415_FB,
  AV_ControlledVariable		:= A_360_01_SK4_A415_C,
  AV_ManualOverride			:= A_360_01_SK4_A415_KMD,
  BV_ExcludeFromOptimizer	:= A_360_01_SK4_A415_OPT_EKSKL,
  BV_DamperError				:= A_360_01_SK4_A415_A1,
  BV_CommunicationError		:= A_360_01_SK4_A415_A2,
  modbusHoldingRegisters		:= ADR(GVL_Modbus.awHoldingRegisters[i * 30]), 
  modbusCoilRegisters			:= ADR(GVL_Modbus.axCoils[i]), 
  typDamperInterface	    :=  GVL_Modbus.ModbusDamperInterface[1][18], 
  typDamperSettings       := PersistentVars.ModbusDamperSetpoints[1][18]
);
i := i +1;
// Kommunikasjonsalarmer

                
// Mappinger for spjeld +A=360.01-SK5A415

bacnetModbusDamperInterop[1][19](
  AI_Volume					:= A_360_01_SK5_A415_VOL,
  AV_CurrentSetpoint			:= A_360_01_SK5_A415_SP,
  AV_vMin					:= A_360_01_SK5_A415_VMIN,
  AV_vMax					:= A_360_01_SK5_A415_VMAX,
  AI_Position				:= A_360_01_SK5_A415_FB,
  AV_ControlledVariable		:= A_360_01_SK5_A415_C,
  AV_ManualOverride			:= A_360_01_SK5_A415_KMD,
  BV_ExcludeFromOptimizer	:= A_360_01_SK5_A415_OPT_EKSKL,
  BV_DamperError				:= A_360_01_SK5_A415_A1,
  BV_CommunicationError		:= A_360_01_SK5_A415_A2,
  modbusHoldingRegisters		:= ADR(GVL_Modbus.awHoldingRegisters[i * 30]), 
  modbusCoilRegisters			:= ADR(GVL_Modbus.axCoils[i]), 
  typDamperInterface	    :=  GVL_Modbus.ModbusDamperInterface[1][19], 
  typDamperSettings       := PersistentVars.ModbusDamperSetpoints[1][19]
);
i := i +1;
// Kommunikasjonsalarmer

                
// Mappinger for spjeld +A=360.01-SK5A418

bacnetModbusDamperInterop[1][20](
  AI_Volume					:= A_360_01_SK5_A418_VOL,
  AV_CurrentSetpoint			:= A_360_01_SK5_A418_SP,
  AV_vMin					:= A_360_01_SK5_A418_VMIN,
  AV_vMax					:= A_360_01_SK5_A418_VMAX,
  AI_Position				:= A_360_01_SK5_A418_FB,
  AV_ControlledVariable		:= A_360_01_SK5_A418_C,
  AV_ManualOverride			:= A_360_01_SK5_A418_KMD,
  BV_ExcludeFromOptimizer	:= A_360_01_SK5_A418_OPT_EKSKL,
  BV_DamperError				:= A_360_01_SK5_A418_A1,
  BV_CommunicationError		:= A_360_01_SK5_A418_A2,
  modbusHoldingRegisters		:= ADR(GVL_Modbus.awHoldingRegisters[i * 30]), 
  modbusCoilRegisters			:= ADR(GVL_Modbus.axCoils[i]), 
  typDamperInterface	    :=  GVL_Modbus.ModbusDamperInterface[1][20], 
  typDamperSettings       := PersistentVars.ModbusDamperSetpoints[1][20]
);
i := i +1;
// Kommunikasjonsalarmer

                
// Mappinger for spjeld +A=360.01-SK4A417

bacnetModbusDamperInterop[1][21](
  AI_Volume					:= A_360_01_SK4_A417_VOL,
  AV_CurrentSetpoint			:= A_360_01_SK4_A417_SP,
  AV_vMin					:= A_360_01_SK4_A417_VMIN,
  AV_vMax					:= A_360_01_SK4_A417_VMAX,
  AI_Position				:= A_360_01_SK4_A417_FB,
  AV_ControlledVariable		:= A_360_01_SK4_A417_C,
  AV_ManualOverride			:= A_360_01_SK4_A417_KMD,
  BV_ExcludeFromOptimizer	:= A_360_01_SK4_A417_OPT_EKSKL,
  BV_DamperError				:= A_360_01_SK4_A417_A1,
  BV_CommunicationError		:= A_360_01_SK4_A417_A2,
  modbusHoldingRegisters		:= ADR(GVL_Modbus.awHoldingRegisters[i * 30]), 
  modbusCoilRegisters			:= ADR(GVL_Modbus.axCoils[i]), 
  typDamperInterface	    :=  GVL_Modbus.ModbusDamperInterface[1][21], 
  typDamperSettings       := PersistentVars.ModbusDamperSetpoints[1][21]
);
i := i +1;
// Kommunikasjonsalarmer

                
// Mappinger for spjeld +A=360.01-SQ5C411

